REGION Network 211: Transfer P&P Left Clamp WORK
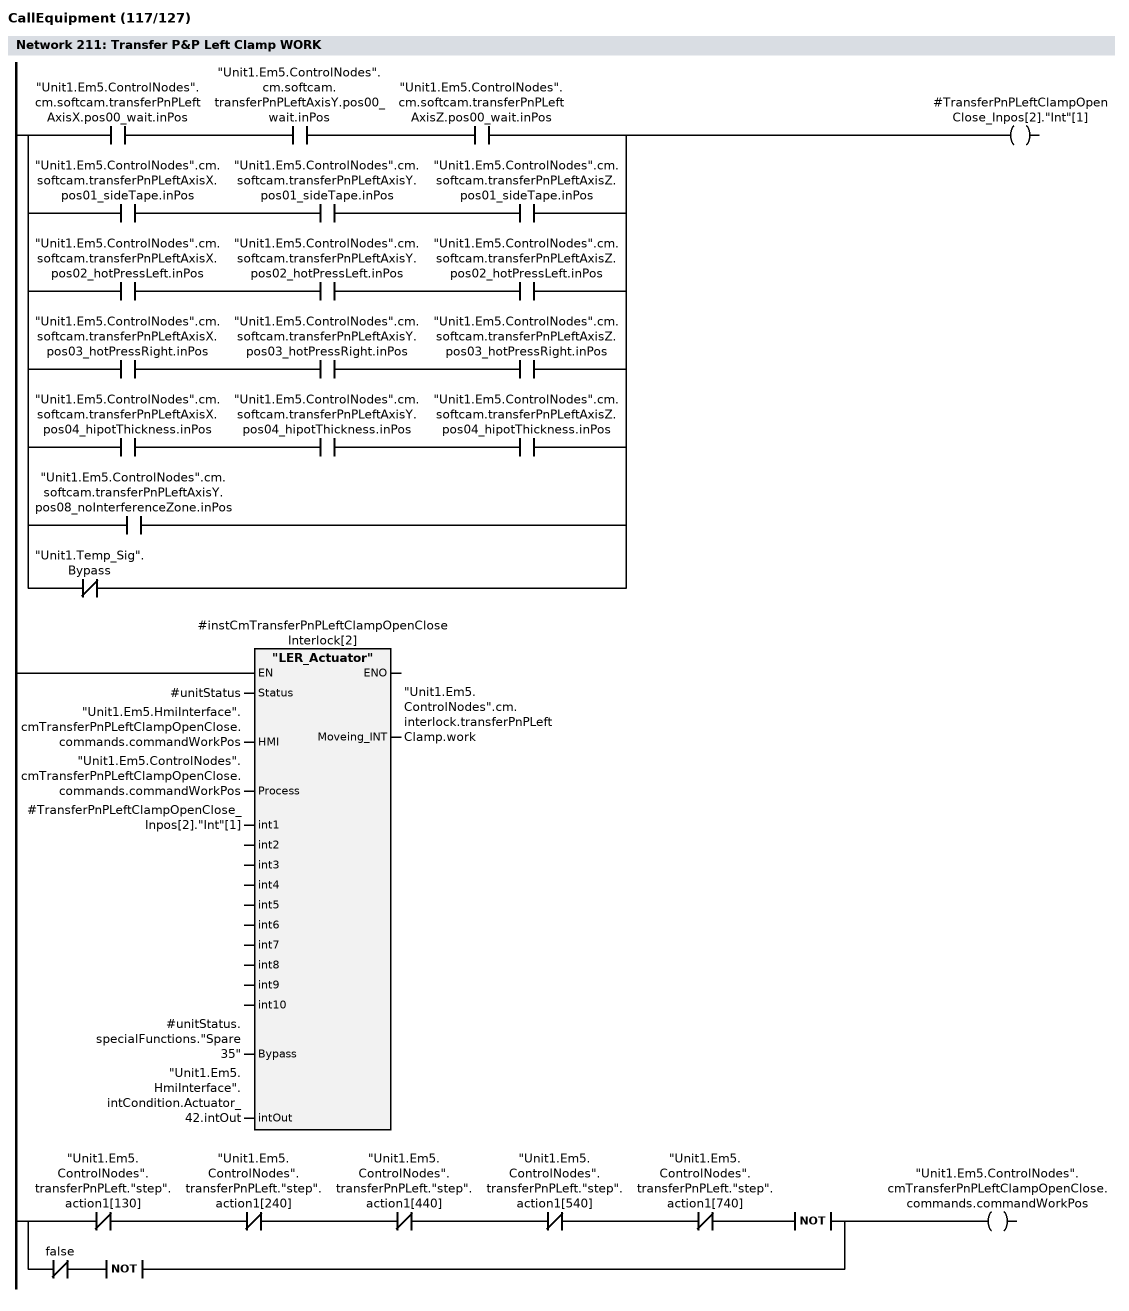
   RUNG wire#powerrail
      Contact( "Unit1.Em5.ControlNodes".cm.softcam.transferPnPLeftAxisX.pos00_wait.inPos )
      Contact( "Unit1.Em5.ControlNodes".cm.softcam.transferPnPLeftAxisY.pos00_wait.inPos )
      Contact( "Unit1.Em5.ControlNodes".cm.softcam.transferPnPLeftAxisZ.pos00_wait.inPos )
      wire#w1
      Coil( #TransferPnPLeftClampOpenClose_Inpos[2]."Int"[1] )
   END_RUNG
   RUNG wire#powerrail
      Contact( "Unit1.Em5.ControlNodes".cm.softcam.transferPnPLeftAxisX.pos01_sideTape.inPos )
      Contact( "Unit1.Em5.ControlNodes".cm.softcam.transferPnPLeftAxisY.pos01_sideTape.inPos )
      Contact( "Unit1.Em5.ControlNodes".cm.softcam.transferPnPLeftAxisZ.pos01_sideTape.inPos )
   END_RUNG wire#w1
   RUNG wire#powerrail
      Contact( "Unit1.Em5.ControlNodes".cm.softcam.transferPnPLeftAxisX.pos02_hotPressLeft.inPos )
      Contact( "Unit1.Em5.ControlNodes".cm.softcam.transferPnPLeftAxisY.pos02_hotPressLeft.inPos )
      Contact( "Unit1.Em5.ControlNodes".cm.softcam.transferPnPLeftAxisZ.pos02_hotPressLeft.inPos )
   END_RUNG wire#w1
   RUNG wire#powerrail
      Contact( "Unit1.Em5.ControlNodes".cm.softcam.transferPnPLeftAxisX.pos03_hotPressRight.inPos )
      Contact( "Unit1.Em5.ControlNodes".cm.softcam.transferPnPLeftAxisY.pos03_hotPressRight.inPos )
      Contact( "Unit1.Em5.ControlNodes".cm.softcam.transferPnPLeftAxisZ.pos03_hotPressRight.inPos )
   END_RUNG wire#w1
   RUNG wire#powerrail
      Contact( "Unit1.Em5.ControlNodes".cm.softcam.transferPnPLeftAxisX.pos04_hipotThickness.inPos )
      Contact( "Unit1.Em5.ControlNodes".cm.softcam.transferPnPLeftAxisY.pos04_hipotThickness.inPos )
      Contact( "Unit1.Em5.ControlNodes".cm.softcam.transferPnPLeftAxisZ.pos04_hipotThickness.inPos )
   END_RUNG wire#w1
   RUNG wire#powerrail
      Contact( "Unit1.Em5.ControlNodes".cm.softcam.transferPnPLeftAxisY.pos08_noInterferenceZone.inPos )
   END_RUNG wire#w1
   RUNG wire#powerrail
      I_Contact( "Unit1.Temp_Sig".Bypass )
   END_RUNG wire#w1
   RUNG wire#powerrail
      #instCmTransferPnPLeftClampOpenCloseInterlock[2](Status := #unitStatus, HMI := "Unit1.Em5.HmiInterface".cmTransferPnPLeftClampOpenClose.commands.commandWorkPos, Process := "Unit1.Em5.ControlNodes".cmTransferPnPLeftClampOpenClose.commands.commandWorkPos, int1 := #TransferPnPLeftClampOpenClose_Inpos[2]."Int"[1], int2 :=, int3 :=, int4 :=, int5 :=, int6 :=, int7 :=, int8 :=, int9 :=, int10 :=, Bypass := #unitStatus.specialFunctions."Spare 35", intOut := "Unit1.Em5.HmiInterface".intCondition.Actuator_42.intOut, Moveing_INT => "Unit1.Em5.ControlNodes".cm.interlock.transferPnPLeftClamp.work)
   END_RUNG
   RUNG wire#powerrail
      I_Contact( "Unit1.Em5.ControlNodes".transferPnPLeft."step".action1[130] )
      I_Contact( "Unit1.Em5.ControlNodes".transferPnPLeft."step".action1[240] )
      I_Contact( "Unit1.Em5.ControlNodes".transferPnPLeft."step".action1[440] )
      I_Contact( "Unit1.Em5.ControlNodes".transferPnPLeft."step".action1[540] )
      I_Contact( "Unit1.Em5.ControlNodes".transferPnPLeft."step".action1[740] )
      Not()
      wire#w2
      Coil( "Unit1.Em5.ControlNodes".cmTransferPnPLeftClampOpenClose.commands.commandWorkPos )
   END_RUNG
   RUNG wire#powerrail
      I_Contact( false )
      Not()
   END_RUNG wire#w2
   // the same network as SCL:
   #TransferPnPLeftClampOpenClose_Inpos[2]."Int"[1] := ("Unit1.Em5.ControlNodes".cm.softcam.transferPnPLeftAxisX.pos00_wait.inPos AND "Unit1.Em5.ControlNodes".cm.softcam.transferPnPLeftAxisY.pos00_wait.inPos AND "Unit1.Em5.ControlNodes".cm.softcam.transferPnPLeftAxisZ.pos00_wait.inPos) OR ("Unit1.Em5.ControlNodes".cm.softcam.transferPnPLeftAxisX.pos01_sideTape.inPos AND "Unit1.Em5.ControlNodes".cm.softcam.transferPnPLeftAxisY.pos01_sideTape.inPos AND "Unit1.Em5.ControlNodes".cm.softcam.transferPnPLeftAxisZ.pos01_sideTape.inPos) OR ("Unit1.Em5.ControlNodes".cm.softcam.transferPnPLeftAxisX.pos02_hotPressLeft.inPos AND "Unit1.Em5.ControlNodes".cm.softcam.transferPnPLeftAxisY.pos02_hotPressLeft.inPos AND "Unit1.Em5.ControlNodes".cm.softcam.transferPnPLeftAxisZ.pos02_hotPressLeft.inPos) OR ("Unit1.Em5.ControlNodes".cm.softcam.transferPnPLeftAxisX.pos03_hotPressRight.inPos AND "Unit1.Em5.ControlNodes".cm.softcam.transferPnPLeftAxisY.pos03_hotPressRight.inPos AND "Unit1.Em5.ControlNodes".cm.softcam.transferPnPLeftAxisZ.pos03_hotPressRight.inPos) OR ("Unit1.Em5.ControlNodes".cm.softcam.transferPnPLeftAxisX.pos04_hipotThickness.inPos AND "Unit1.Em5.ControlNodes".cm.softcam.transferPnPLeftAxisY.pos04_hipotThickness.inPos AND "Unit1.Em5.ControlNodes".cm.softcam.transferPnPLeftAxisZ.pos04_hipotThickness.inPos) OR "Unit1.Em5.ControlNodes".cm.softcam.transferPnPLeftAxisY.pos08_noInterferenceZone.inPos OR NOT "Unit1.Temp_Sig".Bypass;
   #instCmTransferPnPLeftClampOpenCloseInterlock[2](Status := #unitStatus,   // "LER_Actuator"
                           HMI := "Unit1.Em5.HmiInterface".cmTransferPnPLeftClampOpenClose.commands.commandWorkPos,
                           Process := "Unit1.Em5.ControlNodes".cmTransferPnPLeftClampOpenClose.commands.commandWorkPos,
                           int1 := #TransferPnPLeftClampOpenClose_Inpos[2]."Int"[1],
                           Bypass := #unitStatus.specialFunctions."Spare 35",
                           intOut := "Unit1.Em5.HmiInterface".intCondition.Actuator_42.intOut,
                           Moveing_INT => "Unit1.Em5.ControlNodes".cm.interlock.transferPnPLeftClamp.work);
   "Unit1.Em5.ControlNodes".cmTransferPnPLeftClampOpenClose.commands.commandWorkPos := NOT (NOT "Unit1.Em5.ControlNodes".transferPnPLeft."step".action1[130] AND NOT "Unit1.Em5.ControlNodes".transferPnPLeft."step".action1[240] AND NOT "Unit1.Em5.ControlNodes".transferPnPLeft."step".action1[440] AND NOT "Unit1.Em5.ControlNodes".transferPnPLeft."step".action1[540] AND NOT "Unit1.Em5.ControlNodes".transferPnPLeft."step".action1[740]) OR NOT (NOT false);
END_REGION

REGION Network 212: Call CM Transfer P&P Left Clamp Open/Close (LBC_TwoWayActuator)
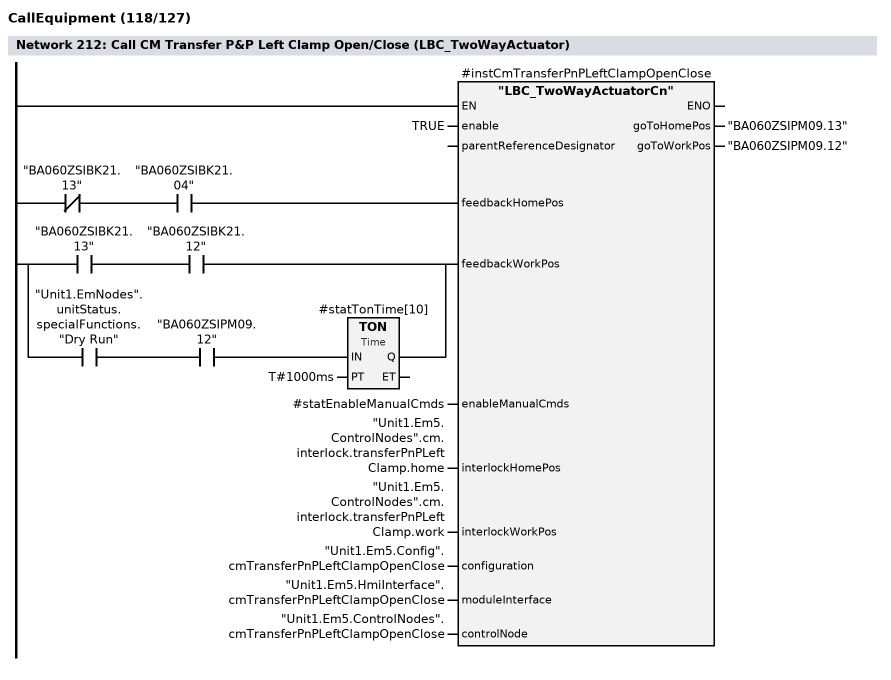
   RUNG wire#powerrail
      #instCmTransferPnPLeftClampOpenClose(feedbackHomePos := wire#w1, feedbackWorkPos := wire#w2, enable := TRUE, parentReferenceDesignator :=, enableManualCmds := #statEnableManualCmds, interlockHomePos := "Unit1.Em5.ControlNodes".cm.interlock.transferPnPLeftClamp.home, interlockWorkPos := "Unit1.Em5.ControlNodes".cm.interlock.transferPnPLeftClamp.work, configuration := "Unit1.Em5.Config".cmTransferPnPLeftClampOpenClose, moduleInterface := "Unit1.Em5.HmiInterface".cmTransferPnPLeftClampOpenClose, controlNode := "Unit1.Em5.ControlNodes".cmTransferPnPLeftClampOpenClose, goToHomePos => "BA060ZSIPM09.13", goToWorkPos => "BA060ZSIPM09.12")
   END_RUNG
   RUNG wire#powerrail
      I_Contact( "BA060ZSIBK21.13" )
      Contact( "BA060ZSIBK21.04" )
   END_RUNG wire#w1
   RUNG wire#powerrail
      Contact( "BA060ZSIBK21.13" )
      Contact( "BA060ZSIBK21.12" )
   END_RUNG wire#w2
   RUNG wire#powerrail
      Contact( "Unit1.EmNodes".unitStatus.specialFunctions."Dry Run" )
      Contact( "BA060ZSIPM09.12" )
      { S7_Templates := "time_type := Time" } #statTonTime[10].TON(pt := T#1000ms, et =>)
   END_RUNG wire#w2
   // the same network as SCL:
   #statTonTime[10].TON(IN := "Unit1.EmNodes".unitStatus.specialFunctions."Dry Run" AND "BA060ZSIPM09.12",
                        PT := T#1000ms);
   #instCmTransferPnPLeftClampOpenClose(enable := TRUE,   // "LBC_TwoWayActuatorCn"
                           feedbackHomePos := NOT "BA060ZSIBK21.13" AND "BA060ZSIBK21.04",
                           feedbackWorkPos := ("BA060ZSIBK21.13" AND "BA060ZSIBK21.12") OR #statTonTime[10].Q,
                           enableManualCmds := #statEnableManualCmds,
                           interlockHomePos := "Unit1.Em5.ControlNodes".cm.interlock.transferPnPLeftClamp.home,
                           interlockWorkPos := "Unit1.Em5.ControlNodes".cm.interlock.transferPnPLeftClamp.work,
                           configuration := "Unit1.Em5.Config".cmTransferPnPLeftClampOpenClose,
                           moduleInterface := "Unit1.Em5.HmiInterface".cmTransferPnPLeftClampOpenClose,
                           controlNode := "Unit1.Em5.ControlNodes".cmTransferPnPLeftClampOpenClose,
                           goToHomePos => "BA060ZSIPM09.13",
                           goToWorkPos => "BA060ZSIPM09.12");
END_REGION

REGION Network 214: Transfer P&P Right Clamp HOME
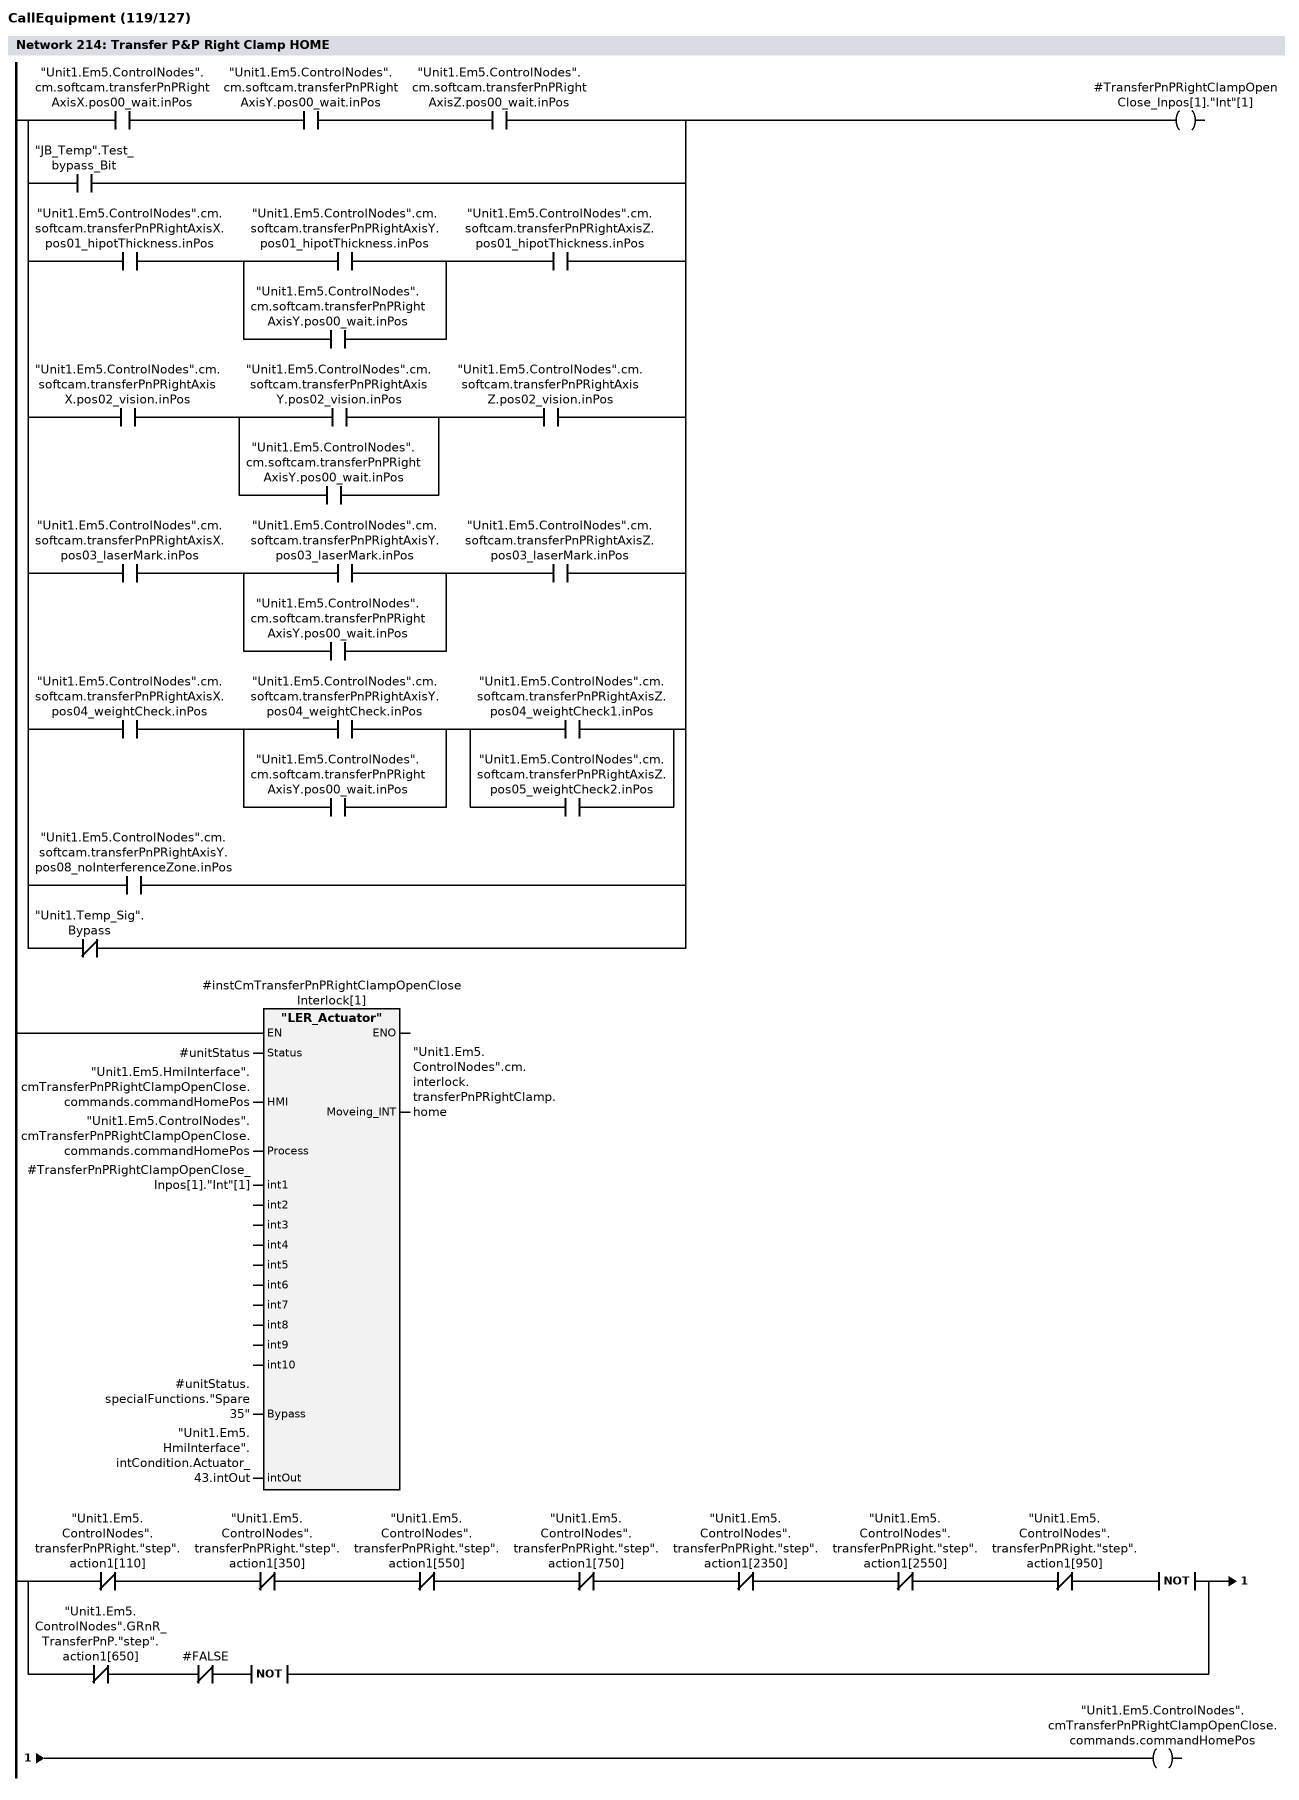
   RUNG wire#powerrail
      Contact( "Unit1.Em5.ControlNodes".cm.softcam.transferPnPRightAxisX.pos00_wait.inPos )
      Contact( "Unit1.Em5.ControlNodes".cm.softcam.transferPnPRightAxisY.pos00_wait.inPos )
      Contact( "Unit1.Em5.ControlNodes".cm.softcam.transferPnPRightAxisZ.pos00_wait.inPos )
      wire#w1
      Coil( #TransferPnPRightClampOpenClose_Inpos[1]."Int"[1] )
   END_RUNG
   RUNG wire#powerrail
      Contact( "JB_Temp".Test_bypass_Bit )
   END_RUNG wire#w1
   RUNG wire#powerrail
      Contact( "Unit1.Em5.ControlNodes".cm.softcam.transferPnPRightAxisX.pos01_hipotThickness.inPos )
      wire#w2
      Contact( "Unit1.Em5.ControlNodes".cm.softcam.transferPnPRightAxisY.pos01_hipotThickness.inPos )
      wire#w3
      Contact( "Unit1.Em5.ControlNodes".cm.softcam.transferPnPRightAxisZ.pos01_hipotThickness.inPos )
   END_RUNG wire#w1
   RUNG wire#w2
      Contact( "Unit1.Em5.ControlNodes".cm.softcam.transferPnPRightAxisY.pos00_wait.inPos )
   END_RUNG wire#w3
   RUNG wire#powerrail
      Contact( "Unit1.Em5.ControlNodes".cm.softcam.transferPnPRightAxisX.pos02_vision.inPos )
      wire#w4
      Contact( "Unit1.Em5.ControlNodes".cm.softcam.transferPnPRightAxisY.pos02_vision.inPos )
      wire#w5
      Contact( "Unit1.Em5.ControlNodes".cm.softcam.transferPnPRightAxisZ.pos02_vision.inPos )
   END_RUNG wire#w1
   RUNG wire#w4
      Contact( "Unit1.Em5.ControlNodes".cm.softcam.transferPnPRightAxisY.pos00_wait.inPos )
   END_RUNG wire#w5
   RUNG wire#powerrail
      Contact( "Unit1.Em5.ControlNodes".cm.softcam.transferPnPRightAxisX.pos03_laserMark.inPos )
      wire#w6
      Contact( "Unit1.Em5.ControlNodes".cm.softcam.transferPnPRightAxisY.pos03_laserMark.inPos )
      wire#w7
      Contact( "Unit1.Em5.ControlNodes".cm.softcam.transferPnPRightAxisZ.pos03_laserMark.inPos )
   END_RUNG wire#w1
   RUNG wire#w6
      Contact( "Unit1.Em5.ControlNodes".cm.softcam.transferPnPRightAxisY.pos00_wait.inPos )
   END_RUNG wire#w7
   RUNG wire#powerrail
      Contact( "Unit1.Em5.ControlNodes".cm.softcam.transferPnPRightAxisX.pos04_weightCheck.inPos )
      wire#w8
      Contact( "Unit1.Em5.ControlNodes".cm.softcam.transferPnPRightAxisY.pos04_weightCheck.inPos )
      wire#w9
      Contact( "Unit1.Em5.ControlNodes".cm.softcam.transferPnPRightAxisZ.pos04_weightCheck1.inPos )
   END_RUNG wire#w1
   RUNG wire#w8
      Contact( "Unit1.Em5.ControlNodes".cm.softcam.transferPnPRightAxisY.pos00_wait.inPos )
   END_RUNG wire#w9
   RUNG wire#w9
      Contact( "Unit1.Em5.ControlNodes".cm.softcam.transferPnPRightAxisZ.pos05_weightCheck2.inPos )
   END_RUNG wire#w1
   RUNG wire#powerrail
      Contact( "Unit1.Em5.ControlNodes".cm.softcam.transferPnPRightAxisY.pos08_noInterferenceZone.inPos )
   END_RUNG wire#w1
   RUNG wire#powerrail
      I_Contact( "Unit1.Temp_Sig".Bypass )
   END_RUNG wire#w1
   RUNG wire#powerrail
      #instCmTransferPnPRightClampOpenCloseInterlock[1](Status := #unitStatus, HMI := "Unit1.Em5.HmiInterface".cmTransferPnPRightClampOpenClose.commands.commandHomePos, Process := "Unit1.Em5.ControlNodes".cmTransferPnPRightClampOpenClose.commands.commandHomePos, int1 := #TransferPnPRightClampOpenClose_Inpos[1]."Int"[1], int2 :=, int3 :=, int4 :=, int5 :=, int6 :=, int7 :=, int8 :=, int9 :=, int10 :=, Bypass := #unitStatus.specialFunctions."Spare 35", intOut := "Unit1.Em5.HmiInterface".intCondition.Actuator_43.intOut, Moveing_INT => "Unit1.Em5.ControlNodes".cm.interlock.transferPnPRightClamp.home)
   END_RUNG
   RUNG wire#powerrail
      I_Contact( "Unit1.Em5.ControlNodes".transferPnPRight."step".action1[110] )
      I_Contact( "Unit1.Em5.ControlNodes".transferPnPRight."step".action1[350] )
      I_Contact( "Unit1.Em5.ControlNodes".transferPnPRight."step".action1[550] )
      I_Contact( "Unit1.Em5.ControlNodes".transferPnPRight."step".action1[750] )
      I_Contact( "Unit1.Em5.ControlNodes".transferPnPRight."step".action1[2350] )
      I_Contact( "Unit1.Em5.ControlNodes".transferPnPRight."step".action1[2550] )
      I_Contact( "Unit1.Em5.ControlNodes".transferPnPRight."step".action1[950] )
      Not()
      wire#w10
      Coil( "Unit1.Em5.ControlNodes".cmTransferPnPRightClampOpenClose.commands.commandHomePos )
   END_RUNG
   RUNG wire#powerrail
      I_Contact( "Unit1.Em5.ControlNodes".GRnR_TransferPnP."step".action1[650] )
      I_Contact( #FALSE )
      Not()
   END_RUNG wire#w10
   // the same network as SCL:
   #TransferPnPRightClampOpenClose_Inpos[1]."Int"[1] := ("Unit1.Em5.ControlNodes".cm.softcam.transferPnPRightAxisX.pos00_wait.inPos AND "Unit1.Em5.ControlNodes".cm.softcam.transferPnPRightAxisY.pos00_wait.inPos AND "Unit1.Em5.ControlNodes".cm.softcam.transferPnPRightAxisZ.pos00_wait.inPos) OR "JB_Temp".Test_bypass_Bit OR ("Unit1.Em5.ControlNodes".cm.softcam.transferPnPRightAxisX.pos01_hipotThickness.inPos AND ("Unit1.Em5.ControlNodes".cm.softcam.transferPnPRightAxisY.pos01_hipotThickness.inPos OR "Unit1.Em5.ControlNodes".cm.softcam.transferPnPRightAxisY.pos00_wait.inPos) AND "Unit1.Em5.ControlNodes".cm.softcam.transferPnPRightAxisZ.pos01_hipotThickness.inPos) OR ("Unit1.Em5.ControlNodes".cm.softcam.transferPnPRightAxisX.pos02_vision.inPos AND ("Unit1.Em5.ControlNodes".cm.softcam.transferPnPRightAxisY.pos02_vision.inPos OR "Unit1.Em5.ControlNodes".cm.softcam.transferPnPRightAxisY.pos00_wait.inPos) AND "Unit1.Em5.ControlNodes".cm.softcam.transferPnPRightAxisZ.pos02_vision.inPos) OR ("Unit1.Em5.ControlNodes".cm.softcam.transferPnPRightAxisX.pos03_laserMark.inPos AND ("Unit1.Em5.ControlNodes".cm.softcam.transferPnPRightAxisY.pos03_laserMark.inPos OR "Unit1.Em5.ControlNodes".cm.softcam.transferPnPRightAxisY.pos00_wait.inPos) AND "Unit1.Em5.ControlNodes".cm.softcam.transferPnPRightAxisZ.pos03_laserMark.inPos) OR ("Unit1.Em5.ControlNodes".cm.softcam.transferPnPRightAxisX.pos04_weightCheck.inPos AND ("Unit1.Em5.ControlNodes".cm.softcam.transferPnPRightAxisY.pos04_weightCheck.inPos OR "Unit1.Em5.ControlNodes".cm.softcam.transferPnPRightAxisY.pos00_wait.inPos) AND ("Unit1.Em5.ControlNodes".cm.softcam.transferPnPRightAxisZ.pos04_weightCheck1.inPos OR "Unit1.Em5.ControlNodes".cm.softcam.transferPnPRightAxisZ.pos05_weightCheck2.inPos)) OR "Unit1.Em5.ControlNodes".cm.softcam.transferPnPRightAxisY.pos08_noInterferenceZone.inPos OR NOT "Unit1.Temp_Sig".Bypass;
   #instCmTransferPnPRightClampOpenCloseInterlock[1](Status := #unitStatus,   // "LER_Actuator"
                           HMI := "Unit1.Em5.HmiInterface".cmTransferPnPRightClampOpenClose.commands.commandHomePos,
                           Process := "Unit1.Em5.ControlNodes".cmTransferPnPRightClampOpenClose.commands.commandHomePos,
                           int1 := #TransferPnPRightClampOpenClose_Inpos[1]."Int"[1],
                           Bypass := #unitStatus.specialFunctions."Spare 35",
                           intOut := "Unit1.Em5.HmiInterface".intCondition.Actuator_43.intOut,
                           Moveing_INT => "Unit1.Em5.ControlNodes".cm.interlock.transferPnPRightClamp.home);
   "Unit1.Em5.ControlNodes".cmTransferPnPRightClampOpenClose.commands.commandHomePos := NOT (NOT "Unit1.Em5.ControlNodes".transferPnPRight."step".action1[110] AND NOT "Unit1.Em5.ControlNodes".transferPnPRight."step".action1[350] AND NOT "Unit1.Em5.ControlNodes".transferPnPRight."step".action1[550] AND NOT "Unit1.Em5.ControlNodes".transferPnPRight."step".action1[750] AND NOT "Unit1.Em5.ControlNodes".transferPnPRight."step".action1[2350] AND NOT "Unit1.Em5.ControlNodes".transferPnPRight."step".action1[2550] AND NOT "Unit1.Em5.ControlNodes".transferPnPRight."step".action1[950]) OR NOT (NOT "Unit1.Em5.ControlNodes".GRnR_TransferPnP."step".action1[650] AND NOT #FALSE);
END_REGION

REGION Network 215: Transfer P&P Right Clamp WORK
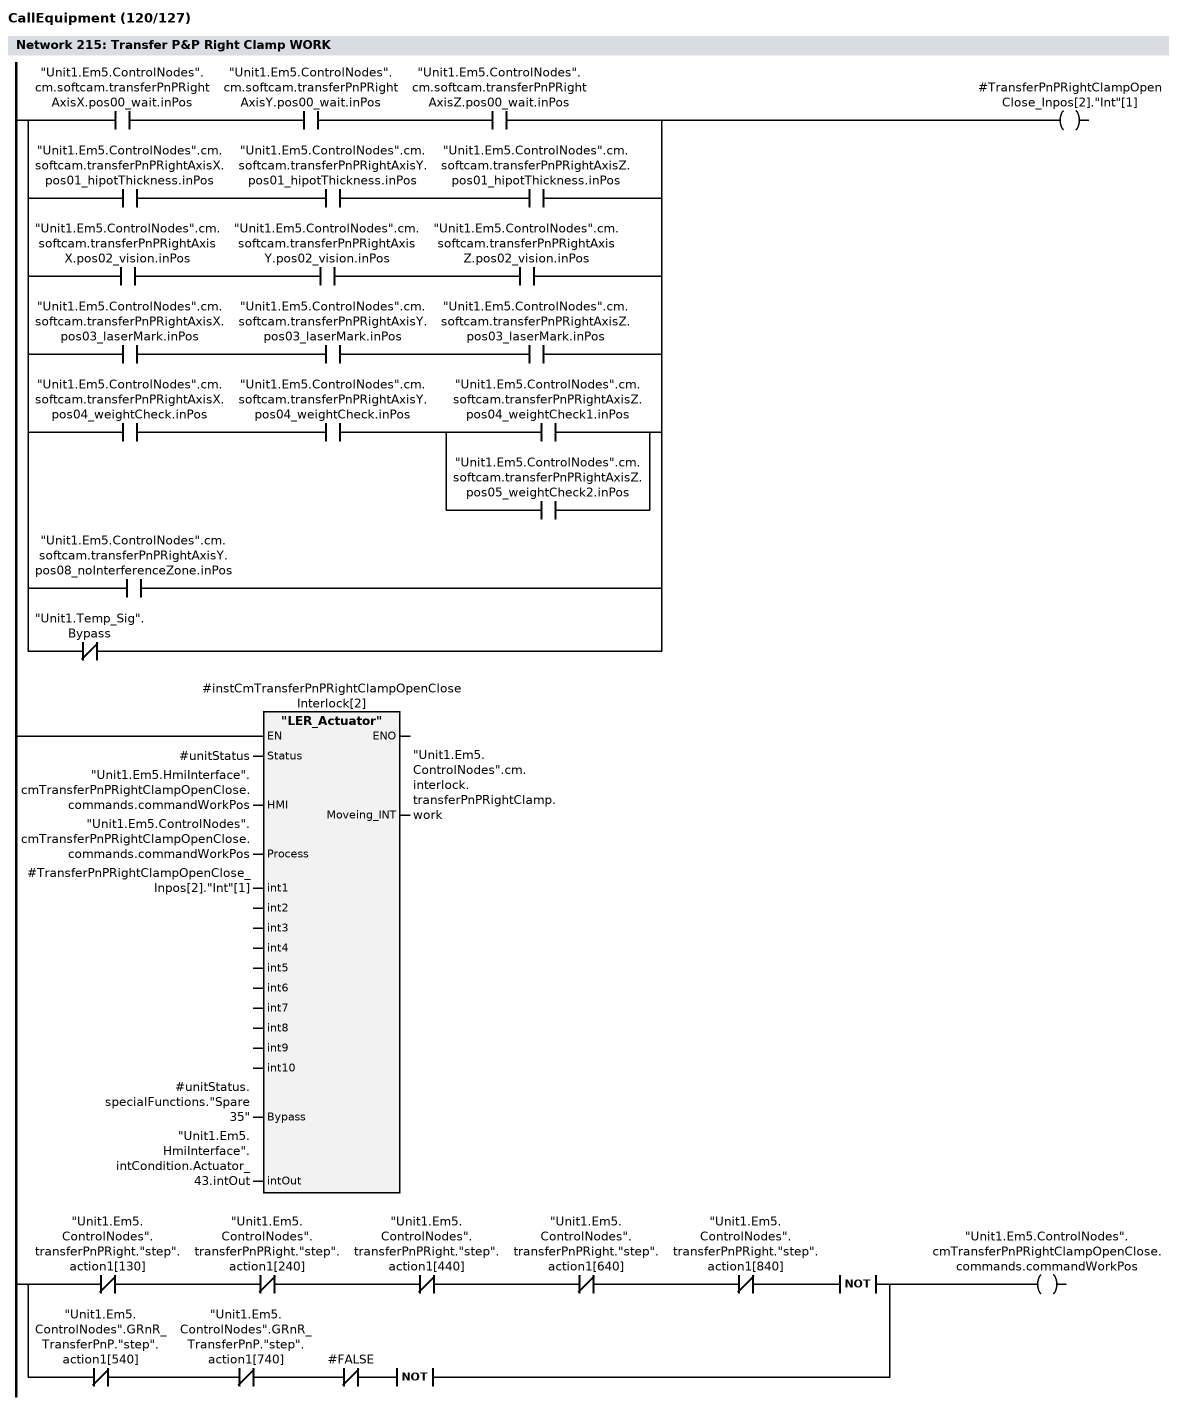
   RUNG wire#powerrail
      Contact( "Unit1.Em5.ControlNodes".cm.softcam.transferPnPRightAxisX.pos00_wait.inPos )
      Contact( "Unit1.Em5.ControlNodes".cm.softcam.transferPnPRightAxisY.pos00_wait.inPos )
      Contact( "Unit1.Em5.ControlNodes".cm.softcam.transferPnPRightAxisZ.pos00_wait.inPos )
      wire#w1
      Coil( #TransferPnPRightClampOpenClose_Inpos[2]."Int"[1] )
   END_RUNG
   RUNG wire#powerrail
      Contact( "Unit1.Em5.ControlNodes".cm.softcam.transferPnPRightAxisX.pos01_hipotThickness.inPos )
      Contact( "Unit1.Em5.ControlNodes".cm.softcam.transferPnPRightAxisY.pos01_hipotThickness.inPos )
      Contact( "Unit1.Em5.ControlNodes".cm.softcam.transferPnPRightAxisZ.pos01_hipotThickness.inPos )
   END_RUNG wire#w1
   RUNG wire#powerrail
      Contact( "Unit1.Em5.ControlNodes".cm.softcam.transferPnPRightAxisX.pos02_vision.inPos )
      Contact( "Unit1.Em5.ControlNodes".cm.softcam.transferPnPRightAxisY.pos02_vision.inPos )
      Contact( "Unit1.Em5.ControlNodes".cm.softcam.transferPnPRightAxisZ.pos02_vision.inPos )
   END_RUNG wire#w1
   RUNG wire#powerrail
      Contact( "Unit1.Em5.ControlNodes".cm.softcam.transferPnPRightAxisX.pos03_laserMark.inPos )
      Contact( "Unit1.Em5.ControlNodes".cm.softcam.transferPnPRightAxisY.pos03_laserMark.inPos )
      Contact( "Unit1.Em5.ControlNodes".cm.softcam.transferPnPRightAxisZ.pos03_laserMark.inPos )
   END_RUNG wire#w1
   RUNG wire#powerrail
      Contact( "Unit1.Em5.ControlNodes".cm.softcam.transferPnPRightAxisX.pos04_weightCheck.inPos )
      Contact( "Unit1.Em5.ControlNodes".cm.softcam.transferPnPRightAxisY.pos04_weightCheck.inPos )
      wire#w2
      Contact( "Unit1.Em5.ControlNodes".cm.softcam.transferPnPRightAxisZ.pos04_weightCheck1.inPos )
   END_RUNG wire#w1
   RUNG wire#w2
      Contact( "Unit1.Em5.ControlNodes".cm.softcam.transferPnPRightAxisZ.pos05_weightCheck2.inPos )
   END_RUNG wire#w1
   RUNG wire#powerrail
      Contact( "Unit1.Em5.ControlNodes".cm.softcam.transferPnPRightAxisY.pos08_noInterferenceZone.inPos )
   END_RUNG wire#w1
   RUNG wire#powerrail
      I_Contact( "Unit1.Temp_Sig".Bypass )
   END_RUNG wire#w1
   RUNG wire#powerrail
      #instCmTransferPnPRightClampOpenCloseInterlock[2](Status := #unitStatus, HMI := "Unit1.Em5.HmiInterface".cmTransferPnPRightClampOpenClose.commands.commandWorkPos, Process := "Unit1.Em5.ControlNodes".cmTransferPnPRightClampOpenClose.commands.commandWorkPos, int1 := #TransferPnPRightClampOpenClose_Inpos[2]."Int"[1], int2 :=, int3 :=, int4 :=, int5 :=, int6 :=, int7 :=, int8 :=, int9 :=, int10 :=, Bypass := #unitStatus.specialFunctions."Spare 35", intOut := "Unit1.Em5.HmiInterface".intCondition.Actuator_43.intOut, Moveing_INT => "Unit1.Em5.ControlNodes".cm.interlock.transferPnPRightClamp.work)
   END_RUNG
   RUNG wire#powerrail
      I_Contact( "Unit1.Em5.ControlNodes".transferPnPRight."step".action1[130] )
      I_Contact( "Unit1.Em5.ControlNodes".transferPnPRight."step".action1[240] )
      I_Contact( "Unit1.Em5.ControlNodes".transferPnPRight."step".action1[440] )
      I_Contact( "Unit1.Em5.ControlNodes".transferPnPRight."step".action1[640] )
      I_Contact( "Unit1.Em5.ControlNodes".transferPnPRight."step".action1[840] )
      Not()
      wire#w3
      Coil( "Unit1.Em5.ControlNodes".cmTransferPnPRightClampOpenClose.commands.commandWorkPos )
   END_RUNG
   RUNG wire#powerrail
      I_Contact( "Unit1.Em5.ControlNodes".GRnR_TransferPnP."step".action1[540] )
      I_Contact( "Unit1.Em5.ControlNodes".GRnR_TransferPnP."step".action1[740] )
      I_Contact( #FALSE )
      Not()
   END_RUNG wire#w3
   // the same network as SCL:
   #TransferPnPRightClampOpenClose_Inpos[2]."Int"[1] := ("Unit1.Em5.ControlNodes".cm.softcam.transferPnPRightAxisX.pos00_wait.inPos AND "Unit1.Em5.ControlNodes".cm.softcam.transferPnPRightAxisY.pos00_wait.inPos AND "Unit1.Em5.ControlNodes".cm.softcam.transferPnPRightAxisZ.pos00_wait.inPos) OR ("Unit1.Em5.ControlNodes".cm.softcam.transferPnPRightAxisX.pos01_hipotThickness.inPos AND "Unit1.Em5.ControlNodes".cm.softcam.transferPnPRightAxisY.pos01_hipotThickness.inPos AND "Unit1.Em5.ControlNodes".cm.softcam.transferPnPRightAxisZ.pos01_hipotThickness.inPos) OR ("Unit1.Em5.ControlNodes".cm.softcam.transferPnPRightAxisX.pos02_vision.inPos AND "Unit1.Em5.ControlNodes".cm.softcam.transferPnPRightAxisY.pos02_vision.inPos AND "Unit1.Em5.ControlNodes".cm.softcam.transferPnPRightAxisZ.pos02_vision.inPos) OR ("Unit1.Em5.ControlNodes".cm.softcam.transferPnPRightAxisX.pos03_laserMark.inPos AND "Unit1.Em5.ControlNodes".cm.softcam.transferPnPRightAxisY.pos03_laserMark.inPos AND "Unit1.Em5.ControlNodes".cm.softcam.transferPnPRightAxisZ.pos03_laserMark.inPos) OR ("Unit1.Em5.ControlNodes".cm.softcam.transferPnPRightAxisX.pos04_weightCheck.inPos AND "Unit1.Em5.ControlNodes".cm.softcam.transferPnPRightAxisY.pos04_weightCheck.inPos AND ("Unit1.Em5.ControlNodes".cm.softcam.transferPnPRightAxisZ.pos04_weightCheck1.inPos OR "Unit1.Em5.ControlNodes".cm.softcam.transferPnPRightAxisZ.pos05_weightCheck2.inPos)) OR "Unit1.Em5.ControlNodes".cm.softcam.transferPnPRightAxisY.pos08_noInterferenceZone.inPos OR NOT "Unit1.Temp_Sig".Bypass;
   #instCmTransferPnPRightClampOpenCloseInterlock[2](Status := #unitStatus,   // "LER_Actuator"
                           HMI := "Unit1.Em5.HmiInterface".cmTransferPnPRightClampOpenClose.commands.commandWorkPos,
                           Process := "Unit1.Em5.ControlNodes".cmTransferPnPRightClampOpenClose.commands.commandWorkPos,
                           int1 := #TransferPnPRightClampOpenClose_Inpos[2]."Int"[1],
                           Bypass := #unitStatus.specialFunctions."Spare 35",
                           intOut := "Unit1.Em5.HmiInterface".intCondition.Actuator_43.intOut,
                           Moveing_INT => "Unit1.Em5.ControlNodes".cm.interlock.transferPnPRightClamp.work);
   "Unit1.Em5.ControlNodes".cmTransferPnPRightClampOpenClose.commands.commandWorkPos := NOT (NOT "Unit1.Em5.ControlNodes".transferPnPRight."step".action1[130] AND NOT "Unit1.Em5.ControlNodes".transferPnPRight."step".action1[240] AND NOT "Unit1.Em5.ControlNodes".transferPnPRight."step".action1[440] AND NOT "Unit1.Em5.ControlNodes".transferPnPRight."step".action1[640] AND NOT "Unit1.Em5.ControlNodes".transferPnPRight."step".action1[840]) OR NOT (NOT "Unit1.Em5.ControlNodes".GRnR_TransferPnP."step".action1[540] AND NOT "Unit1.Em5.ControlNodes".GRnR_TransferPnP."step".action1[740] AND NOT #FALSE);
END_REGION

REGION Network 216: Call CM Transfer P&P Right Clamp Open/Close (LBC_TwoWayActuator)
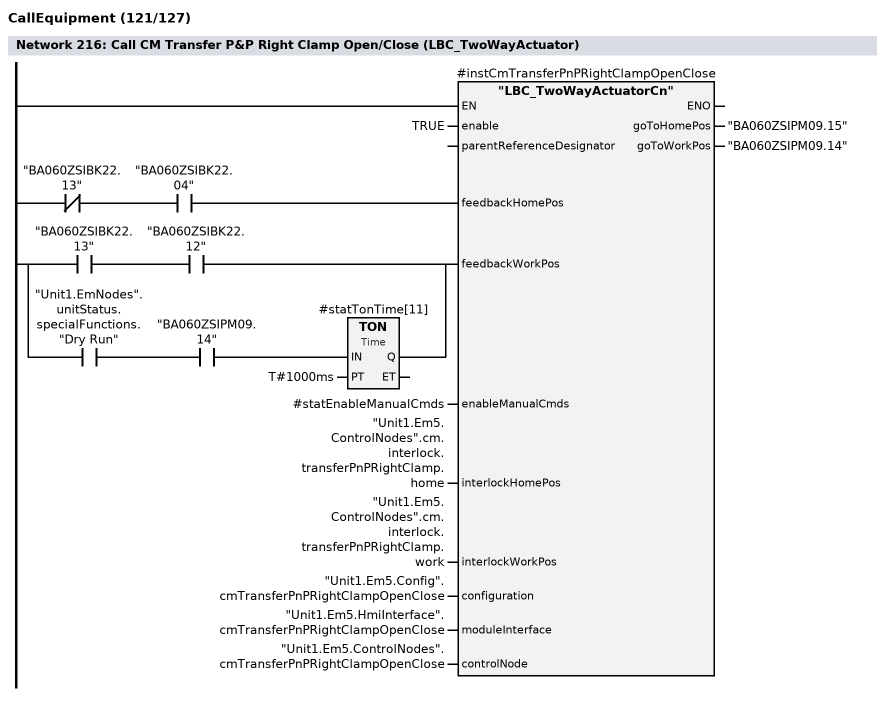
   RUNG wire#powerrail
      #instCmTransferPnPRightClampOpenClose(feedbackHomePos := wire#w1, feedbackWorkPos := wire#w2, enable := TRUE, parentReferenceDesignator :=, enableManualCmds := #statEnableManualCmds, interlockHomePos := "Unit1.Em5.ControlNodes".cm.interlock.transferPnPRightClamp.home, interlockWorkPos := "Unit1.Em5.ControlNodes".cm.interlock.transferPnPRightClamp.work, configuration := "Unit1.Em5.Config".cmTransferPnPRightClampOpenClose, moduleInterface := "Unit1.Em5.HmiInterface".cmTransferPnPRightClampOpenClose, controlNode := "Unit1.Em5.ControlNodes".cmTransferPnPRightClampOpenClose, goToHomePos => "BA060ZSIPM09.15", goToWorkPos => "BA060ZSIPM09.14")
   END_RUNG
   RUNG wire#powerrail
      I_Contact( "BA060ZSIBK22.13" )
      Contact( "BA060ZSIBK22.04" )
   END_RUNG wire#w1
   RUNG wire#powerrail
      Contact( "BA060ZSIBK22.13" )
      Contact( "BA060ZSIBK22.12" )
   END_RUNG wire#w2
   RUNG wire#powerrail
      Contact( "Unit1.EmNodes".unitStatus.specialFunctions."Dry Run" )
      Contact( "BA060ZSIPM09.14" )
      { S7_Templates := "time_type := Time" } #statTonTime[11].TON(pt := T#1000ms, et =>)
   END_RUNG wire#w2
   // the same network as SCL:
   #statTonTime[11].TON(IN := "Unit1.EmNodes".unitStatus.specialFunctions."Dry Run" AND "BA060ZSIPM09.14",
                        PT := T#1000ms);
   #instCmTransferPnPRightClampOpenClose(enable := TRUE,   // "LBC_TwoWayActuatorCn"
                           feedbackHomePos := NOT "BA060ZSIBK22.13" AND "BA060ZSIBK22.04",
                           feedbackWorkPos := ("BA060ZSIBK22.13" AND "BA060ZSIBK22.12") OR #statTonTime[11].Q,
                           enableManualCmds := #statEnableManualCmds,
                           interlockHomePos := "Unit1.Em5.ControlNodes".cm.interlock.transferPnPRightClamp.home,
                           interlockWorkPos := "Unit1.Em5.ControlNodes".cm.interlock.transferPnPRightClamp.work,
                           configuration := "Unit1.Em5.Config".cmTransferPnPRightClampOpenClose,
                           moduleInterface := "Unit1.Em5.HmiInterface".cmTransferPnPRightClampOpenClose,
                           controlNode := "Unit1.Em5.ControlNodes".cmTransferPnPRightClampOpenClose,
                           goToHomePos => "BA060ZSIPM09.15",
                           goToWorkPos => "BA060ZSIPM09.14");
END_REGION

REGION Network 218: ******************** Feedback to Unit ********************
END_REGION

REGION Network 219: Determine StateComplete (SC) in Mode Production
   // Conditions for the Equipment Modules "stateComplete" feedback to the unit. This feedback is given when the task in for the respective state is complete.
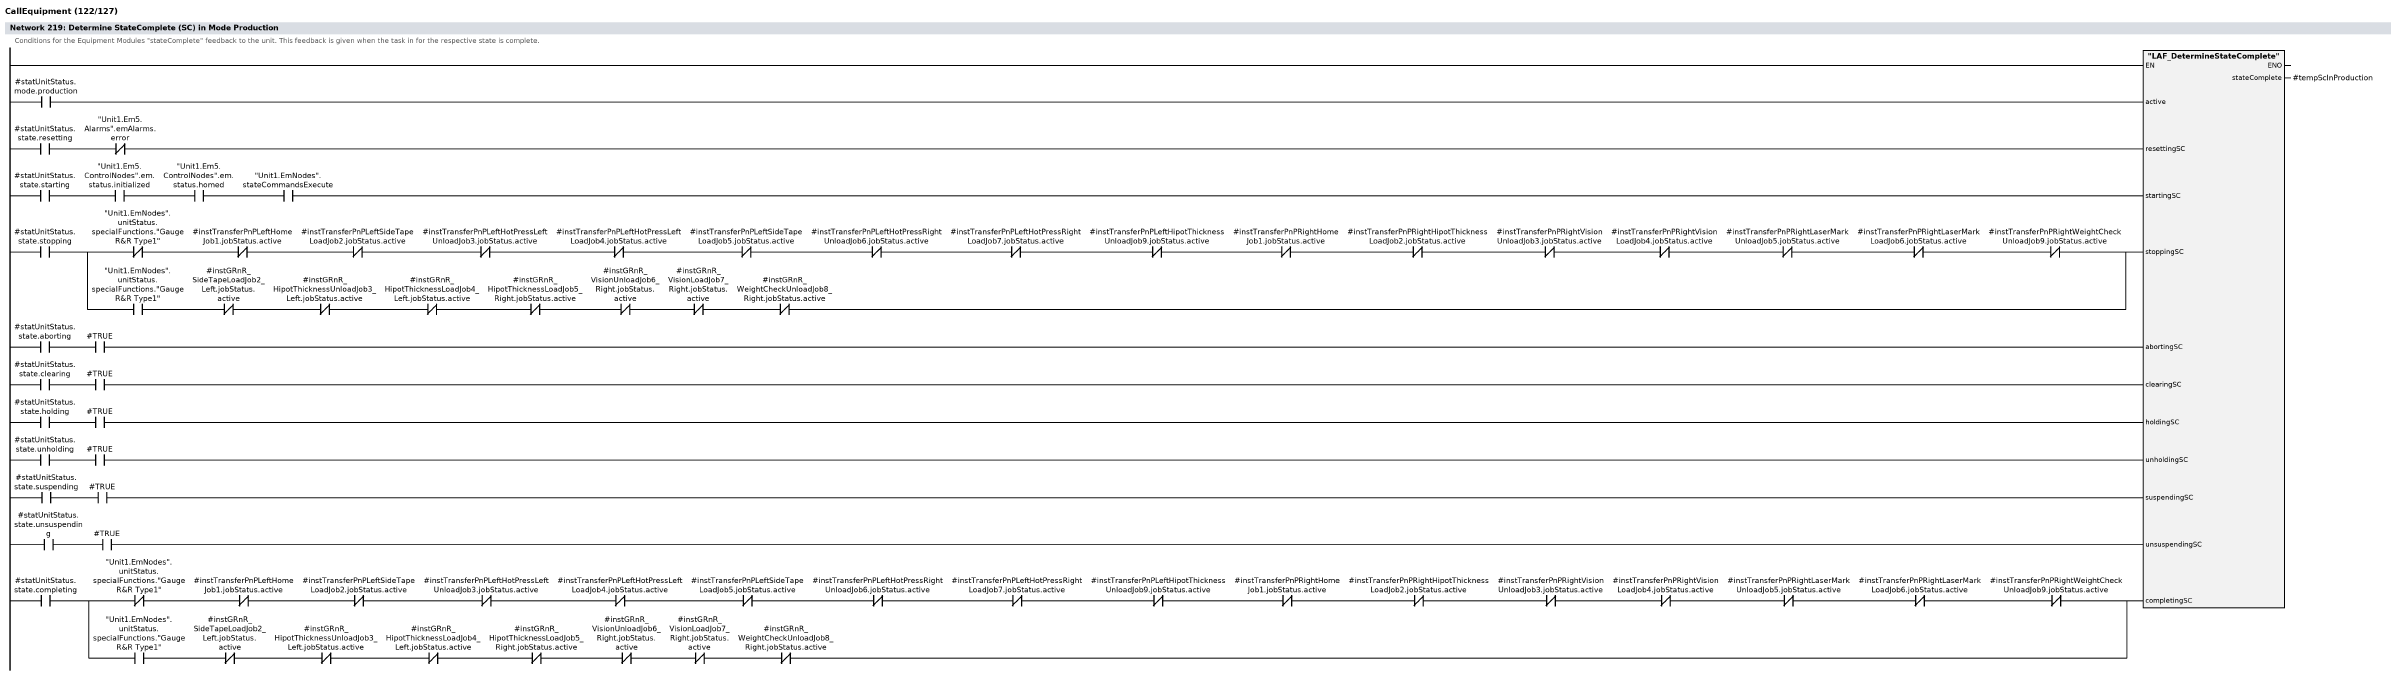
   RUNG wire#powerrail
      "LAF_DetermineStateComplete"(active := wire#w1, resettingSC := wire#w2, startingSC := wire#w3, stoppingSC := wire#w5, abortingSC := wire#w6, clearingSC := wire#w7, holdingSC := wire#w8, unholdingSC := wire#w9, suspendingSC := wire#w10, unsuspendingSC := wire#w11, completingSC := wire#w13, stateComplete => #tempScInProduction)
   END_RUNG
   RUNG wire#powerrail
      Contact( #statUnitStatus.mode.production )
   END_RUNG wire#w1
   RUNG wire#powerrail
      Contact( #statUnitStatus.state.resetting )
      I_Contact( "Unit1.Em5.Alarms".emAlarms.error )
   END_RUNG wire#w2
   RUNG wire#powerrail
      Contact( #statUnitStatus.state.starting )
      Contact( "Unit1.Em5.ControlNodes".em.status.initialized )
      Contact( "Unit1.Em5.ControlNodes".em.status.homed )
      Contact( "Unit1.EmNodes".stateCommandsExecute )
   END_RUNG wire#w3
   RUNG wire#powerrail
      Contact( #statUnitStatus.state.stopping )
      wire#w4
      I_Contact( "Unit1.EmNodes".unitStatus.specialFunctions."Gauge R&R Type1" )
      I_Contact( #instTransferPnPLeftHomeJob1.jobStatus.active )
      I_Contact( #instTransferPnPLeftSideTapeLoadJob2.jobStatus.active )
      I_Contact( #instTransferPnPLeftHotPressLeftUnloadJob3.jobStatus.active )
      I_Contact( #instTransferPnPLeftHotPressLeftLoadJob4.jobStatus.active )
      I_Contact( #instTransferPnPLeftSideTapeLoadJob5.jobStatus.active )
      I_Contact( #instTransferPnPLeftHotPressRightUnloadJob6.jobStatus.active )
      I_Contact( #instTransferPnPLeftHotPressRightLoadJob7.jobStatus.active )
      I_Contact( #instTransferPnPLeftHipotThicknessUnloadJob9.jobStatus.active )
      I_Contact( #instTransferPnPRightHomeJob1.jobStatus.active )
      I_Contact( #instTransferPnPRightHipotThicknessLoadJob2.jobStatus.active )
      I_Contact( #instTransferPnPRightVisionUnloadJob3.jobStatus.active )
      I_Contact( #instTransferPnPRightVisionLoadJob4.jobStatus.active )
      I_Contact( #instTransferPnPRightLaserMarkUnloadJob5.jobStatus.active )
      I_Contact( #instTransferPnPRightLaserMarkLoadJob6.jobStatus.active )
      I_Contact( #instTransferPnPRightWeightCheckUnloadJob9.jobStatus.active )
   END_RUNG wire#w5
   RUNG wire#w4
      Contact( "Unit1.EmNodes".unitStatus.specialFunctions."Gauge R&R Type1" )
      I_Contact( #instGRnR_SideTapeLoadJob2_Left.jobStatus.active )
      I_Contact( #instGRnR_HipotThicknessUnloadJob3_Left.jobStatus.active )
      I_Contact( #instGRnR_HipotThicknessLoadJob4_Left.jobStatus.active )
      I_Contact( #instGRnR_HipotThicknessLoadJob5_Right.jobStatus.active )
      I_Contact( #instGRnR_VisionUnloadJob6_Right.jobStatus.active )
      I_Contact( #instGRnR_VisionLoadJob7_Right.jobStatus.active )
      I_Contact( #instGRnR_WeightCheckUnloadJob8_Right.jobStatus.active )
   END_RUNG wire#w5
   RUNG wire#powerrail
      Contact( #statUnitStatus.state.aborting )
      Contact( #TRUE )
   END_RUNG wire#w6
   RUNG wire#powerrail
      Contact( #statUnitStatus.state.clearing )
      Contact( #TRUE )
   END_RUNG wire#w7
   RUNG wire#powerrail
      Contact( #statUnitStatus.state.holding )
      Contact( #TRUE )
   END_RUNG wire#w8
   RUNG wire#powerrail
      Contact( #statUnitStatus.state.unholding )
      Contact( #TRUE )
   END_RUNG wire#w9
   RUNG wire#powerrail
      Contact( #statUnitStatus.state.suspending )
      Contact( #TRUE )
   END_RUNG wire#w10
   RUNG wire#powerrail
      Contact( #statUnitStatus.state.unsuspending )
      Contact( #TRUE )
   END_RUNG wire#w11
   RUNG wire#powerrail
      Contact( #statUnitStatus.state.completing )
      wire#w12
      I_Contact( "Unit1.EmNodes".unitStatus.specialFunctions."Gauge R&R Type1" )
      I_Contact( #instTransferPnPLeftHomeJob1.jobStatus.active )
      I_Contact( #instTransferPnPLeftSideTapeLoadJob2.jobStatus.active )
      I_Contact( #instTransferPnPLeftHotPressLeftUnloadJob3.jobStatus.active )
      I_Contact( #instTransferPnPLeftHotPressLeftLoadJob4.jobStatus.active )
      I_Contact( #instTransferPnPLeftSideTapeLoadJob5.jobStatus.active )
      I_Contact( #instTransferPnPLeftHotPressRightUnloadJob6.jobStatus.active )
      I_Contact( #instTransferPnPLeftHotPressRightLoadJob7.jobStatus.active )
      I_Contact( #instTransferPnPLeftHipotThicknessUnloadJob9.jobStatus.active )
      I_Contact( #instTransferPnPRightHomeJob1.jobStatus.active )
      I_Contact( #instTransferPnPRightHipotThicknessLoadJob2.jobStatus.active )
      I_Contact( #instTransferPnPRightVisionUnloadJob3.jobStatus.active )
      I_Contact( #instTransferPnPRightVisionLoadJob4.jobStatus.active )
      I_Contact( #instTransferPnPRightLaserMarkUnloadJob5.jobStatus.active )
      I_Contact( #instTransferPnPRightLaserMarkLoadJob6.jobStatus.active )
      I_Contact( #instTransferPnPRightWeightCheckUnloadJob9.jobStatus.active )
   END_RUNG wire#w13
   RUNG wire#w12
      Contact( "Unit1.EmNodes".unitStatus.specialFunctions."Gauge R&R Type1" )
      I_Contact( #instGRnR_SideTapeLoadJob2_Left.jobStatus.active )
      I_Contact( #instGRnR_HipotThicknessUnloadJob3_Left.jobStatus.active )
      I_Contact( #instGRnR_HipotThicknessLoadJob4_Left.jobStatus.active )
      I_Contact( #instGRnR_HipotThicknessLoadJob5_Right.jobStatus.active )
      I_Contact( #instGRnR_VisionUnloadJob6_Right.jobStatus.active )
      I_Contact( #instGRnR_VisionLoadJob7_Right.jobStatus.active )
      I_Contact( #instGRnR_WeightCheckUnloadJob8_Right.jobStatus.active )
   END_RUNG wire#w13
   // the same network as SCL:
   "LAF_DetermineStateComplete"(active := #statUnitStatus.mode.production,
                           resettingSC := #statUnitStatus.state.resetting AND NOT "Unit1.Em5.Alarms".emAlarms.error,
                           startingSC := #statUnitStatus.state.starting AND "Unit1.Em5.ControlNodes".em.status.initialized AND "Unit1.Em5.ControlNodes".em.status.homed AND "Unit1.EmNodes".stateCommandsExecute,
                           stoppingSC := #statUnitStatus.state.stopping AND ((NOT "Unit1.EmNodes".unitStatus.specialFunctions."Gauge R&R Type1" AND NOT #instTransferPnPLeftHomeJob1.jobStatus.active AND NOT #instTransferPnPLeftSideTapeLoadJob2.jobStatus.active AND NOT #instTransferPnPLeftHotPressLeftUnloadJob3.jobStatus.active AND NOT #instTransferPnPLeftHotPressLeftLoadJob4.jobStatus.active AND NOT #instTransferPnPLeftSideTapeLoadJob5.jobStatus.active AND NOT #instTransferPnPLeftHotPressRightUnloadJob6.jobStatus.active AND NOT #instTransferPnPLeftHotPressRightLoadJob7.jobStatus.active AND NOT #instTransferPnPLeftHipotThicknessUnloadJob9.jobStatus.active AND NOT #instTransferPnPRightHomeJob1.jobStatus.active AND NOT #instTransferPnPRightHipotThicknessLoadJob2.jobStatus.active AND NOT #instTransferPnPRightVisionUnloadJob3.jobStatus.active AND NOT #instTransferPnPRightVisionLoadJob4.jobStatus.active AND NOT #instTransferPnPRightLaserMarkUnloadJob5.jobStatus.active AND NOT #instTransferPnPRightLaserMarkLoadJob6.jobStatus.active AND NOT #instTransferPnPRightWeightCheckUnloadJob9.jobStatus.active) OR ("Unit1.EmNodes".unitStatus.specialFunctions."Gauge R&R Type1" AND NOT #instGRnR_SideTapeLoadJob2_Left.jobStatus.active AND NOT #instGRnR_HipotThicknessUnloadJob3_Left.jobStatus.active AND NOT #instGRnR_HipotThicknessLoadJob4_Left.jobStatus.active AND NOT #instGRnR_HipotThicknessLoadJob5_Right.jobStatus.active AND NOT #instGRnR_VisionUnloadJob6_Right.jobStatus.active AND NOT #instGRnR_VisionLoadJob7_Right.jobStatus.active AND NOT #instGRnR_WeightCheckUnloadJob8_Right.jobStatus.active)),
                           abortingSC := #statUnitStatus.state.aborting AND #TRUE,
                           clearingSC := #statUnitStatus.state.clearing AND #TRUE,
                           holdingSC := #statUnitStatus.state.holding AND #TRUE,
                           unholdingSC := #statUnitStatus.state.unholding AND #TRUE,
                           suspendingSC := #statUnitStatus.state.suspending AND #TRUE,
                           unsuspendingSC := #statUnitStatus.state.unsuspending AND #TRUE,
                           completingSC := #statUnitStatus.state.completing AND ((NOT "Unit1.EmNodes".unitStatus.specialFunctions."Gauge R&R Type1" AND NOT #instTransferPnPLeftHomeJob1.jobStatus.active AND NOT #instTransferPnPLeftSideTapeLoadJob2.jobStatus.active AND NOT #instTransferPnPLeftHotPressLeftUnloadJob3.jobStatus.active AND NOT #instTransferPnPLeftHotPressLeftLoadJob4.jobStatus.active AND NOT #instTransferPnPLeftSideTapeLoadJob5.jobStatus.active AND NOT #instTransferPnPLeftHotPressRightUnloadJob6.jobStatus.active AND NOT #instTransferPnPLeftHotPressRightLoadJob7.jobStatus.active AND NOT #instTransferPnPLeftHipotThicknessUnloadJob9.jobStatus.active AND NOT #instTransferPnPRightHomeJob1.jobStatus.active AND NOT #instTransferPnPRightHipotThicknessLoadJob2.jobStatus.active AND NOT #instTransferPnPRightVisionUnloadJob3.jobStatus.active AND NOT #instTransferPnPRightVisionLoadJob4.jobStatus.active AND NOT #instTransferPnPRightLaserMarkUnloadJob5.jobStatus.active AND NOT #instTransferPnPRightLaserMarkLoadJob6.jobStatus.active AND NOT #instTransferPnPRightWeightCheckUnloadJob9.jobStatus.active) OR ("Unit1.EmNodes".unitStatus.specialFunctions."Gauge R&R Type1" AND NOT #instGRnR_SideTapeLoadJob2_Left.jobStatus.active AND NOT #instGRnR_HipotThicknessUnloadJob3_Left.jobStatus.active AND NOT #instGRnR_HipotThicknessLoadJob4_Left.jobStatus.active AND NOT #instGRnR_HipotThicknessLoadJob5_Right.jobStatus.active AND NOT #instGRnR_VisionUnloadJob6_Right.jobStatus.active AND NOT #instGRnR_VisionLoadJob7_Right.jobStatus.active AND NOT #instGRnR_WeightCheckUnloadJob8_Right.jobStatus.active)),
                           stateComplete => #tempScInProduction);
END_REGION

REGION Network 220: Determine StateComplete (SC) in Mode Maintenance/Manual
   // Conditions for the Equipment Modules "stateComplete" feedback to the unit. This feedback is given when the task in for the respective state is complete.
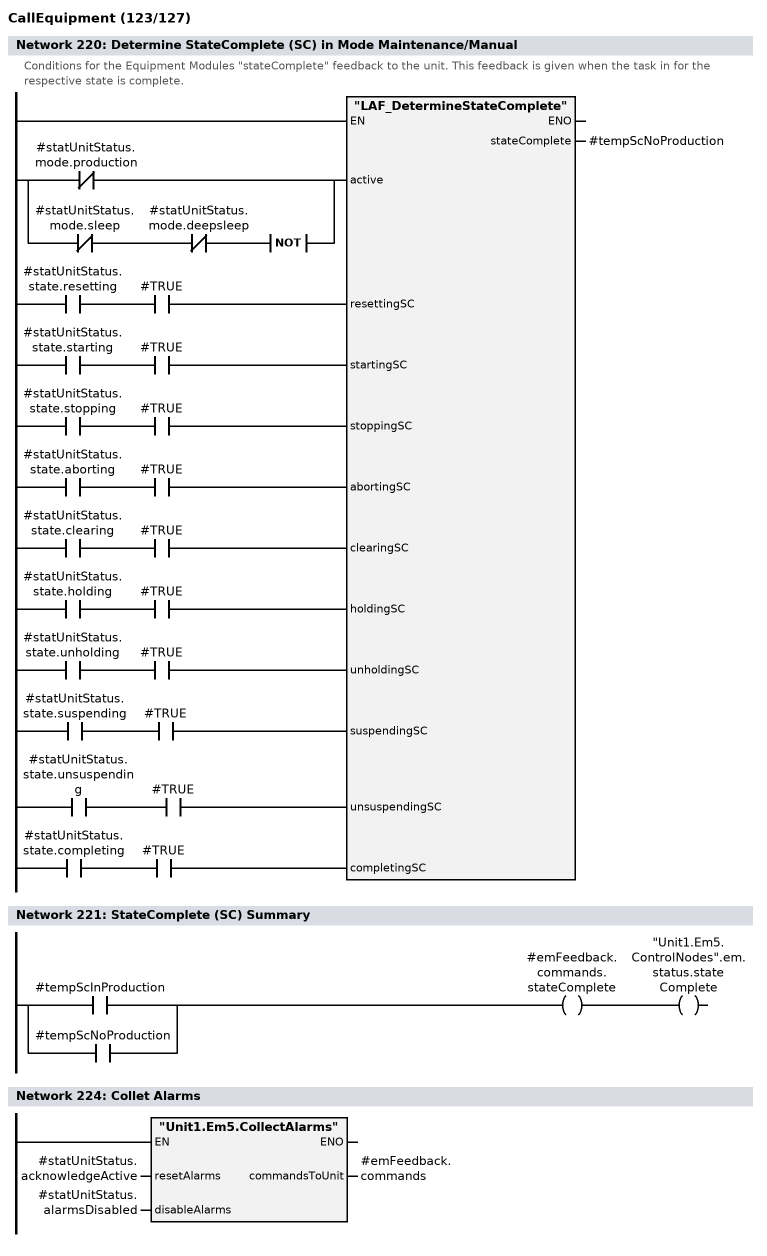
   RUNG wire#powerrail
      "LAF_DetermineStateComplete"(active := wire#w1, resettingSC := wire#w2, startingSC := wire#w3, stoppingSC := wire#w4, abortingSC := wire#w5, clearingSC := wire#w6, holdingSC := wire#w7, unholdingSC := wire#w8, suspendingSC := wire#w9, unsuspendingSC := wire#w10, completingSC := wire#w11, stateComplete => #tempScNoProduction)
   END_RUNG
   RUNG wire#powerrail
      I_Contact( #statUnitStatus.mode.production )
   END_RUNG wire#w1
   RUNG wire#powerrail
      I_Contact( #statUnitStatus.mode.sleep )
      I_Contact( #statUnitStatus.mode.deepsleep )
      Not()
   END_RUNG wire#w1
   RUNG wire#powerrail
      Contact( #statUnitStatus.state.resetting )
      Contact( #TRUE )
   END_RUNG wire#w2
   RUNG wire#powerrail
      Contact( #statUnitStatus.state.starting )
      Contact( #TRUE )
   END_RUNG wire#w3
   RUNG wire#powerrail
      Contact( #statUnitStatus.state.stopping )
      Contact( #TRUE )
   END_RUNG wire#w4
   RUNG wire#powerrail
      Contact( #statUnitStatus.state.aborting )
      Contact( #TRUE )
   END_RUNG wire#w5
   RUNG wire#powerrail
      Contact( #statUnitStatus.state.clearing )
      Contact( #TRUE )
   END_RUNG wire#w6
   RUNG wire#powerrail
      Contact( #statUnitStatus.state.holding )
      Contact( #TRUE )
   END_RUNG wire#w7
   RUNG wire#powerrail
      Contact( #statUnitStatus.state.unholding )
      Contact( #TRUE )
   END_RUNG wire#w8
   RUNG wire#powerrail
      Contact( #statUnitStatus.state.suspending )
      Contact( #TRUE )
   END_RUNG wire#w9
   RUNG wire#powerrail
      Contact( #statUnitStatus.state.unsuspending )
      Contact( #TRUE )
   END_RUNG wire#w10
   RUNG wire#powerrail
      Contact( #statUnitStatus.state.completing )
      Contact( #TRUE )
   END_RUNG wire#w11
   // the same network as SCL:
   "LAF_DetermineStateComplete"(active := NOT #statUnitStatus.mode.production OR NOT (NOT #statUnitStatus.mode.sleep AND NOT #statUnitStatus.mode.deepsleep),
                           resettingSC := #statUnitStatus.state.resetting AND #TRUE,
                           startingSC := #statUnitStatus.state.starting AND #TRUE,
                           stoppingSC := #statUnitStatus.state.stopping AND #TRUE,
                           abortingSC := #statUnitStatus.state.aborting AND #TRUE,
                           clearingSC := #statUnitStatus.state.clearing AND #TRUE,
                           holdingSC := #statUnitStatus.state.holding AND #TRUE,
                           unholdingSC := #statUnitStatus.state.unholding AND #TRUE,
                           suspendingSC := #statUnitStatus.state.suspending AND #TRUE,
                           unsuspendingSC := #statUnitStatus.state.unsuspending AND #TRUE,
                           completingSC := #statUnitStatus.state.completing AND #TRUE,
                           stateComplete => #tempScNoProduction);
END_REGION

REGION Network 221: StateComplete (SC) Summary
   RUNG wire#powerrail
      Contact( #tempScInProduction )
      wire#w1
      Coil( #emFeedback.commands.stateComplete )
      Coil( "Unit1.Em5.ControlNodes".em.status.stateComplete )
   END_RUNG
   RUNG wire#powerrail
      Contact( #tempScNoProduction )
   END_RUNG wire#w1
   // the same network as SCL:
   #emFeedback.commands.stateComplete := #tempScInProduction OR #tempScNoProduction;
   "Unit1.Em5.ControlNodes".em.status.stateComplete := #emFeedback.commands.stateComplete;
END_REGION

REGION Network 223: ******************** Alarms ********************
END_REGION

REGION Network 224: Collet Alarms
   RUNG wire#powerrail
      "Unit1.Em5.CollectAlarms"(resetAlarms := #statUnitStatus.acknowledgeActive, disableAlarms := #statUnitStatus.alarmsDisabled, commandsToUnit => #emFeedback.commands)
   END_RUNG
   // the same network as SCL:
   "Unit1.Em5.CollectAlarms"(resetAlarms := #statUnitStatus.acknowledgeActive,
                           disableAlarms := #statUnitStatus.alarmsDisabled,
                           commandsToUnit => #emFeedback.commands);
END_REGION

REGION Network 225: Manage Alarms
   // Derive commands from the ProDiag supervision. The ProDiag supervisions contain categories which define the reaction of these supervisions (e.g. abort, stop, hold). These are handed over as commands to the unit level.
   // Alternatively, if no ProDiag should be used, you can use the LAF_ManageBitAlarms to realize bit alarm handling. This block can be found in LAF in folder 70_AlarmHandling.
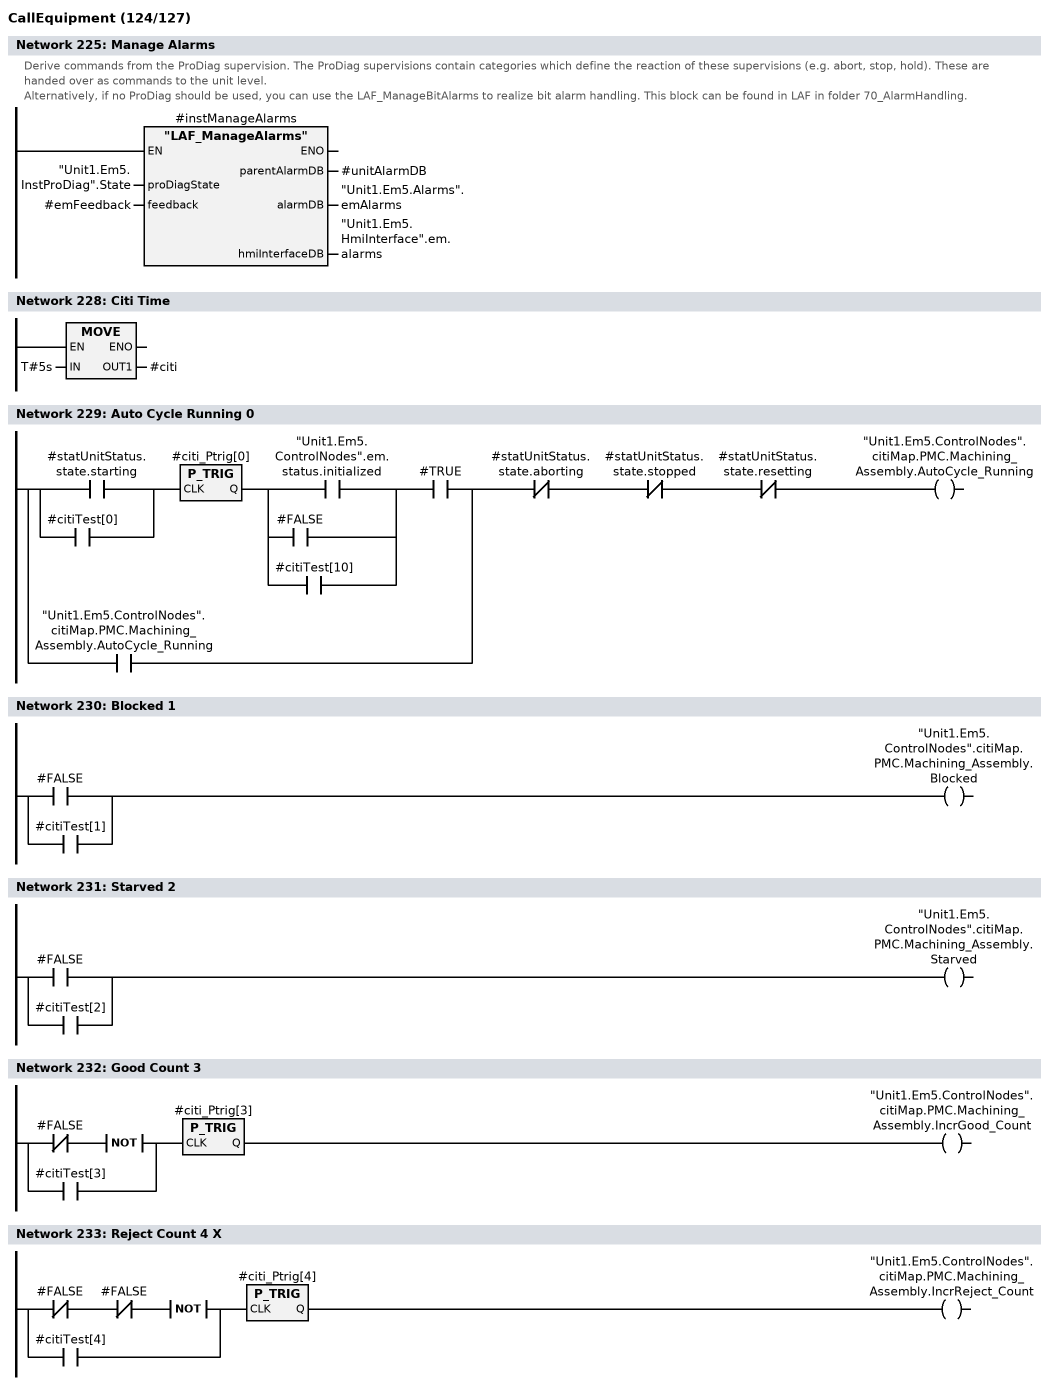
   RUNG wire#powerrail
      #instManageAlarms(proDiagState := "Unit1.Em5.InstProDiag".State, feedback := #emFeedback, parentAlarmDB => #unitAlarmDB, alarmDB => "Unit1.Em5.Alarms".emAlarms, hmiInterfaceDB => "Unit1.Em5.HmiInterface".em.alarms)
   END_RUNG
   // the same network as SCL:
   #instManageAlarms(proDiagState := "Unit1.Em5.InstProDiag".State,   // "LAF_ManageAlarms"
                     feedback := #emFeedback,
                     parentAlarmDB => #unitAlarmDB,
                     alarmDB => "Unit1.Em5.Alarms".emAlarms,
                     hmiInterfaceDB => "Unit1.Em5.HmiInterface".em.alarms);
END_REGION

REGION Network 227: ******************** CITI ********************
END_REGION

REGION Network 228: Citi Time
   RUNG wire#powerrail
      Move(in := T#5s, out1 => #citi)
   END_RUNG
   // the same network as SCL:
   #citi := T#5s;
END_REGION

REGION Network 229: Auto Cycle Running 0
   RUNG wire#powerrail
      Contact( #statUnitStatus.state.starting )
      wire#w1
      P_Trig( #citi_Ptrig[0] )
      wire#w2
      Contact( "Unit1.Em5.ControlNodes".em.status.initialized )
      wire#w3
      Contact( #TRUE )
      wire#w4
      I_Contact( #statUnitStatus.state.aborting )
      I_Contact( #statUnitStatus.state.stopped )
      I_Contact( #statUnitStatus.state.resetting )
      Coil( "Unit1.Em5.ControlNodes".citiMap.PMC.Machining_Assembly.AutoCycle_Running )
   END_RUNG
   RUNG wire#powerrail
      Contact( #citiTest[0] )
   END_RUNG wire#w1
   RUNG wire#w2
      Contact( #FALSE )
   END_RUNG wire#w3
   RUNG wire#w2
      Contact( #citiTest[10] )
   END_RUNG wire#w3
   RUNG wire#powerrail
      Contact( "Unit1.Em5.ControlNodes".citiMap.PMC.Machining_Assembly.AutoCycle_Running )
   END_RUNG wire#w4
   // the same network as SCL:
   #_w1 := #statUnitStatus.state.starting OR #citiTest[0];
   #_w2 := #_w1 AND NOT #citi_Ptrig[0];   // rising edge
   #citi_Ptrig[0] := #_w1;
   "Unit1.Em5.ControlNodes".citiMap.PMC.Machining_Assembly.AutoCycle_Running := ((#_w2 AND ("Unit1.Em5.ControlNodes".em.status.initialized OR #FALSE OR #citiTest[10]) AND #TRUE) OR "Unit1.Em5.ControlNodes".citiMap.PMC.Machining_Assembly.AutoCycle_Running) AND NOT #statUnitStatus.state.aborting AND NOT #statUnitStatus.state.stopped AND NOT #statUnitStatus.state.resetting;
END_REGION

REGION Network 230: Blocked 1
   RUNG wire#powerrail
      Contact( #FALSE )
      wire#w1
      Coil( "Unit1.Em5.ControlNodes".citiMap.PMC.Machining_Assembly.Blocked )
   END_RUNG
   RUNG wire#powerrail
      Contact( #citiTest[1] )
   END_RUNG wire#w1
   // the same network as SCL:
   "Unit1.Em5.ControlNodes".citiMap.PMC.Machining_Assembly.Blocked := #FALSE OR #citiTest[1];
END_REGION

REGION Network 231: Starved 2
   RUNG wire#powerrail
      Contact( #FALSE )
      wire#w1
      Coil( "Unit1.Em5.ControlNodes".citiMap.PMC.Machining_Assembly.Starved )
   END_RUNG
   RUNG wire#powerrail
      Contact( #citiTest[2] )
   END_RUNG wire#w1
   // the same network as SCL:
   "Unit1.Em5.ControlNodes".citiMap.PMC.Machining_Assembly.Starved := #FALSE OR #citiTest[2];
END_REGION

REGION Network 232: Good Count 3
   RUNG wire#powerrail
      I_Contact( #FALSE )
      Not()
      wire#w1
      P_Trig( #citi_Ptrig[3] )
      Coil( "Unit1.Em5.ControlNodes".citiMap.PMC.Machining_Assembly.IncrGood_Count )
   END_RUNG
   RUNG wire#powerrail
      Contact( #citiTest[3] )
   END_RUNG wire#w1
   // the same network as SCL:
   #_w1 := NOT (NOT #FALSE) OR #citiTest[3];
   #_w2 := #_w1 AND NOT #citi_Ptrig[3];   // rising edge
   #citi_Ptrig[3] := #_w1;
   "Unit1.Em5.ControlNodes".citiMap.PMC.Machining_Assembly.IncrGood_Count := #_w2;
END_REGION

REGION Network 233: Reject Count 4 X
   RUNG wire#powerrail
      I_Contact( #FALSE )
      I_Contact( #FALSE )
      Not()
      wire#w1
      P_Trig( #citi_Ptrig[4] )
      Coil( "Unit1.Em5.ControlNodes".citiMap.PMC.Machining_Assembly.IncrReject_Count )
   END_RUNG
   RUNG wire#powerrail
      Contact( #citiTest[4] )
   END_RUNG wire#w1
   // the same network as SCL:
   #_w1 := NOT (NOT #FALSE AND NOT #FALSE) OR #citiTest[4];
   #_w2 := #_w1 AND NOT #citi_Ptrig[4];   // rising edge
   #citi_Ptrig[4] := #_w1;
   "Unit1.Em5.ControlNodes".citiMap.PMC.Machining_Assembly.IncrReject_Count := #_w2;
END_REGION

REGION Network 234: Cycle End Trigger 5
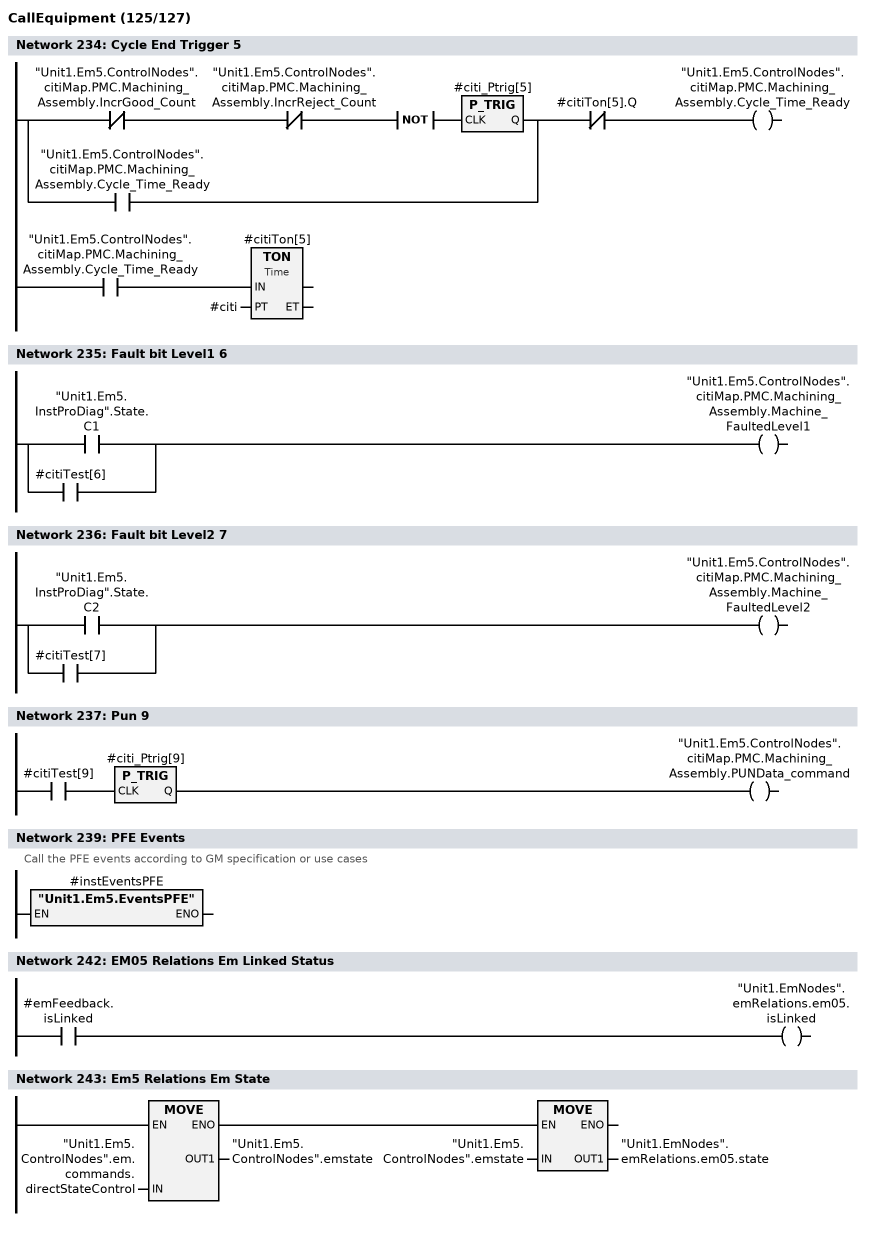
   RUNG wire#powerrail
      I_Contact( "Unit1.Em5.ControlNodes".citiMap.PMC.Machining_Assembly.IncrGood_Count )
      I_Contact( "Unit1.Em5.ControlNodes".citiMap.PMC.Machining_Assembly.IncrReject_Count )
      Not()
      P_Trig( #citi_Ptrig[5] )
      wire#w1
      I_Contact( #citiTon[5].Q )
      Coil( "Unit1.Em5.ControlNodes".citiMap.PMC.Machining_Assembly.Cycle_Time_Ready )
   END_RUNG
   RUNG wire#powerrail
      Contact( "Unit1.Em5.ControlNodes".citiMap.PMC.Machining_Assembly.Cycle_Time_Ready )
   END_RUNG wire#w1
   RUNG wire#powerrail
      Contact( "Unit1.Em5.ControlNodes".citiMap.PMC.Machining_Assembly.Cycle_Time_Ready )
      { S7_Templates := "time_type := Time" } #citiTon[5].TON(pt := #citi, et =>)
   END_RUNG
   // the same network as SCL:
   #_w1 := NOT (NOT "Unit1.Em5.ControlNodes".citiMap.PMC.Machining_Assembly.IncrGood_Count AND NOT "Unit1.Em5.ControlNodes".citiMap.PMC.Machining_Assembly.IncrReject_Count);
   #_w2 := #_w1 AND NOT #citi_Ptrig[5];   // rising edge
   #citi_Ptrig[5] := #_w1;
   "Unit1.Em5.ControlNodes".citiMap.PMC.Machining_Assembly.Cycle_Time_Ready := (#_w2 OR "Unit1.Em5.ControlNodes".citiMap.PMC.Machining_Assembly.Cycle_Time_Ready) AND NOT #citiTon[5].Q;
   #citiTon[5].TON(IN := "Unit1.Em5.ControlNodes".citiMap.PMC.Machining_Assembly.Cycle_Time_Ready, PT := #citi);
END_REGION

REGION Network 235: Fault bit Level1 6
   RUNG wire#powerrail
      Contact( "Unit1.Em5.InstProDiag".State.C1 )
      wire#w1
      Coil( "Unit1.Em5.ControlNodes".citiMap.PMC.Machining_Assembly.Machine_FaultedLevel1 )
   END_RUNG
   RUNG wire#powerrail
      Contact( #citiTest[6] )
   END_RUNG wire#w1
   // the same network as SCL:
   "Unit1.Em5.ControlNodes".citiMap.PMC.Machining_Assembly.Machine_FaultedLevel1 := "Unit1.Em5.InstProDiag".State.C1 OR #citiTest[6];
END_REGION

REGION Network 236: Fault bit Level2 7
   RUNG wire#powerrail
      Contact( "Unit1.Em5.InstProDiag".State.C2 )
      wire#w1
      Coil( "Unit1.Em5.ControlNodes".citiMap.PMC.Machining_Assembly.Machine_FaultedLevel2 )
   END_RUNG
   RUNG wire#powerrail
      Contact( #citiTest[7] )
   END_RUNG wire#w1
   // the same network as SCL:
   "Unit1.Em5.ControlNodes".citiMap.PMC.Machining_Assembly.Machine_FaultedLevel2 := "Unit1.Em5.InstProDiag".State.C2 OR #citiTest[7];
END_REGION

REGION Network 237: Pun 9
   RUNG wire#powerrail
      Contact( #citiTest[9] )
      P_Trig( #citi_Ptrig[9] )
      Coil( "Unit1.Em5.ControlNodes".citiMap.PMC.Machining_Assembly.PUNData_command )
   END_RUNG
   // the same network as SCL:
   #_w1 := #citiTest[9] AND NOT #citi_Ptrig[9];   // rising edge
   #citi_Ptrig[9] := #citiTest[9];
   "Unit1.Em5.ControlNodes".citiMap.PMC.Machining_Assembly.PUNData_command := #_w1;
END_REGION

REGION Network 238: ******************** PFE Events ********************
END_REGION

REGION Network 239: PFE Events
   // Call the PFE events according to GM specification or use cases
   RUNG wire#powerrail
      #instEventsPFE()
   END_RUNG
   // the same network as SCL:
   #instEventsPFE();   // "Unit1.Em5.EventsPFE"
END_REGION

REGION Network 241: ******************** Unit Output ********************
END_REGION

REGION Network 242: EM05 Relations Em Linked Status
   RUNG wire#powerrail
      Contact( #emFeedback.isLinked )
      Coil( "Unit1.EmNodes".emRelations.em05.isLinked )
   END_RUNG
   // the same network as SCL:
   "Unit1.EmNodes".emRelations.em05.isLinked := #emFeedback.isLinked;
END_REGION

REGION Network 243: Em5 Relations Em State
   RUNG wire#powerrail
      Move(in := "Unit1.Em5.ControlNodes".em.commands.directStateControl, out1 => "Unit1.Em5.ControlNodes".emstate)
      Move(in := "Unit1.Em5.ControlNodes".emstate, out1 => "Unit1.EmNodes".emRelations.em05.state)
   END_RUNG
   // the same network as SCL:
   "Unit1.Em5.ControlNodes".emstate := "Unit1.Em5.ControlNodes".em.commands.directStateControl;
   "Unit1.EmNodes".emRelations.em05.state := "Unit1.Em5.ControlNodes".emstate;
END_REGION

REGION Network 244: Em5 User define
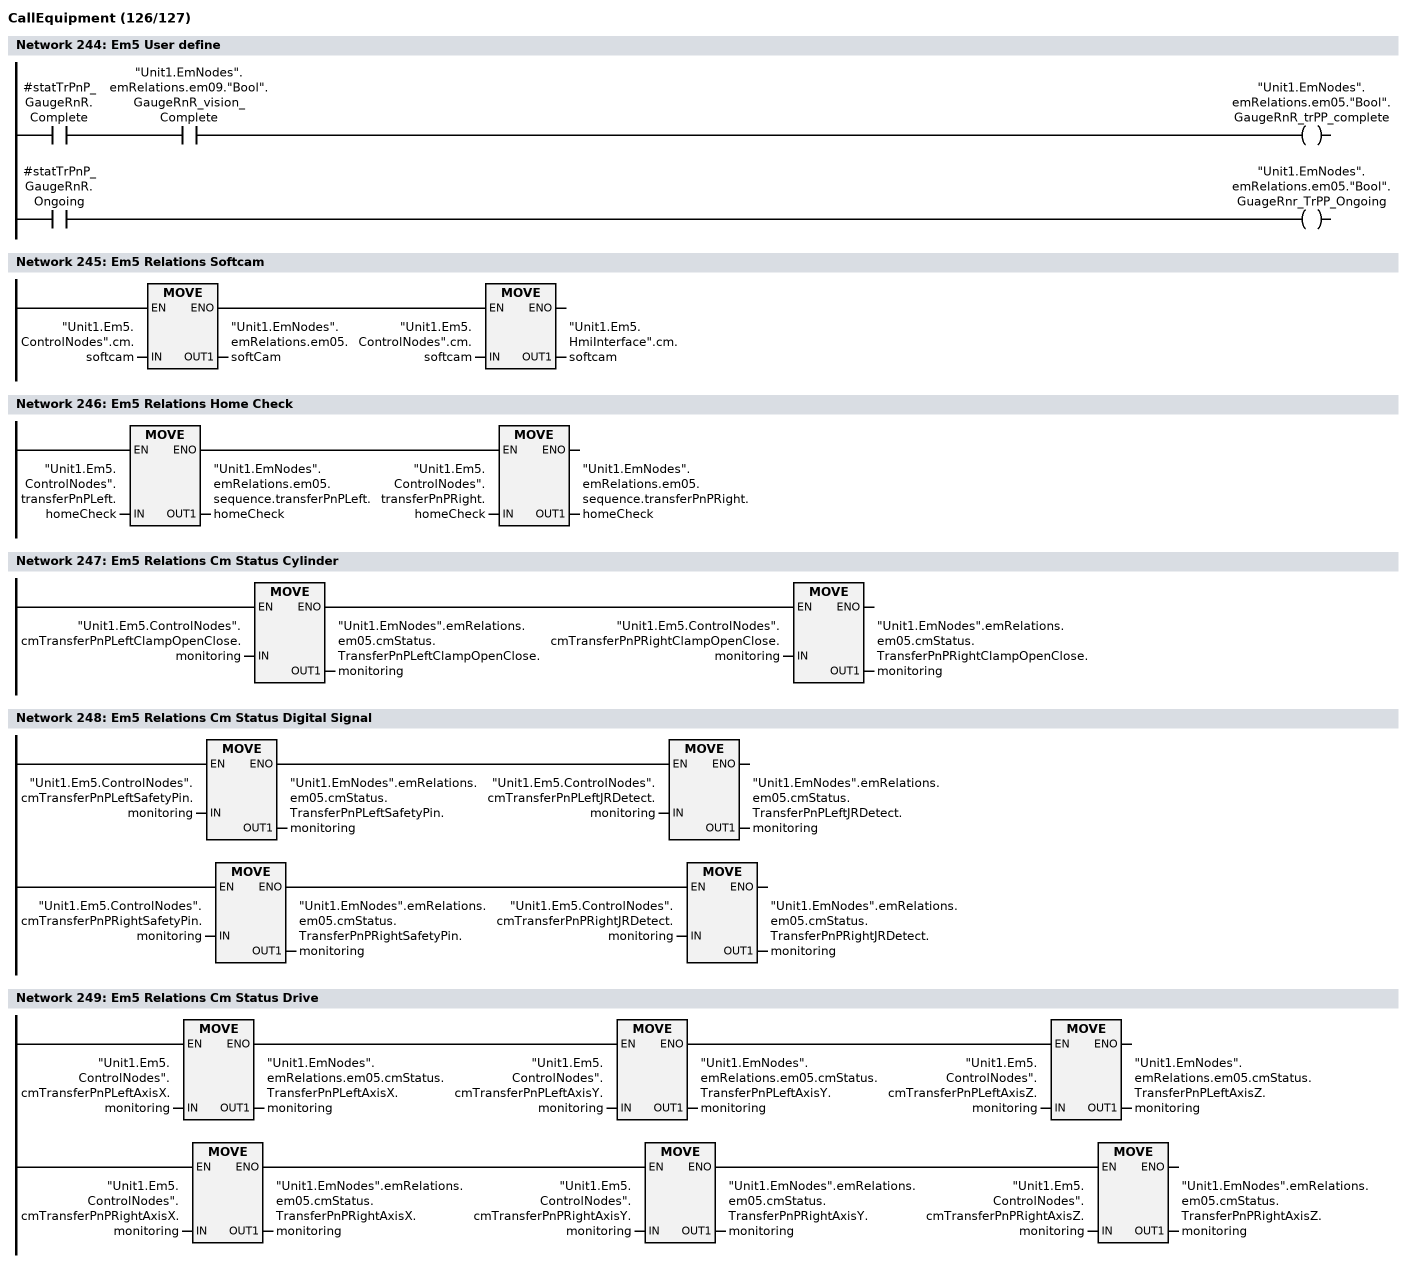
   RUNG wire#powerrail
      Contact( #statTrPnP_GaugeRnR.Complete )
      Contact( "Unit1.EmNodes".emRelations.em09."Bool".GaugeRnR_vision_Complete )
      Coil( "Unit1.EmNodes".emRelations.em05."Bool".GaugeRnR_trPP_complete )
   END_RUNG
   RUNG wire#powerrail
      Contact( #statTrPnP_GaugeRnR.Ongoing )
      Coil( "Unit1.EmNodes".emRelations.em05."Bool".GuageRnr_TrPP_Ongoing )
   END_RUNG
   // the same network as SCL:
   "Unit1.EmNodes".emRelations.em05."Bool".GaugeRnR_trPP_complete := #statTrPnP_GaugeRnR.Complete AND "Unit1.EmNodes".emRelations.em09."Bool".GaugeRnR_vision_Complete;
   "Unit1.EmNodes".emRelations.em05."Bool".GuageRnr_TrPP_Ongoing := #statTrPnP_GaugeRnR.Ongoing;
END_REGION

REGION Network 245: Em5 Relations Softcam
   RUNG wire#powerrail
      Move(in := "Unit1.Em5.ControlNodes".cm.softcam, out1 => "Unit1.EmNodes".emRelations.em05.softCam)
      Move(in := "Unit1.Em5.ControlNodes".cm.softcam, out1 => "Unit1.Em5.HmiInterface".cm.softcam)
   END_RUNG
   // the same network as SCL:
   "Unit1.EmNodes".emRelations.em05.softCam := "Unit1.Em5.ControlNodes".cm.softcam;
   "Unit1.Em5.HmiInterface".cm.softcam := "Unit1.Em5.ControlNodes".cm.softcam;
END_REGION

REGION Network 246: Em5 Relations Home Check
   RUNG wire#powerrail
      Move(in := "Unit1.Em5.ControlNodes".transferPnPLeft.homeCheck, out1 => "Unit1.EmNodes".emRelations.em05.sequence.transferPnPLeft.homeCheck)
      Move(in := "Unit1.Em5.ControlNodes".transferPnPRight.homeCheck, out1 => "Unit1.EmNodes".emRelations.em05.sequence.transferPnPRight.homeCheck)
   END_RUNG
   // the same network as SCL:
   "Unit1.EmNodes".emRelations.em05.sequence.transferPnPLeft.homeCheck := "Unit1.Em5.ControlNodes".transferPnPLeft.homeCheck;
   "Unit1.EmNodes".emRelations.em05.sequence.transferPnPRight.homeCheck := "Unit1.Em5.ControlNodes".transferPnPRight.homeCheck;
END_REGION

REGION Network 247: Em5 Relations Cm Status Cylinder
   RUNG wire#powerrail
      Move(in := "Unit1.Em5.ControlNodes".cmTransferPnPLeftClampOpenClose.monitoring, out1 => "Unit1.EmNodes".emRelations.em05.cmStatus.TransferPnPLeftClampOpenClose.monitoring)
      Move(in := "Unit1.Em5.ControlNodes".cmTransferPnPRightClampOpenClose.monitoring, out1 => "Unit1.EmNodes".emRelations.em05.cmStatus.TransferPnPRightClampOpenClose.monitoring)
   END_RUNG
   // the same network as SCL:
   "Unit1.EmNodes".emRelations.em05.cmStatus.TransferPnPLeftClampOpenClose.monitoring := "Unit1.Em5.ControlNodes".cmTransferPnPLeftClampOpenClose.monitoring;
   "Unit1.EmNodes".emRelations.em05.cmStatus.TransferPnPRightClampOpenClose.monitoring := "Unit1.Em5.ControlNodes".cmTransferPnPRightClampOpenClose.monitoring;
END_REGION

REGION Network 248: Em5 Relations Cm Status Digital Signal
   RUNG wire#powerrail
      Move(in := "Unit1.Em5.ControlNodes".cmTransferPnPLeftSafetyPin.monitoring, out1 => "Unit1.EmNodes".emRelations.em05.cmStatus.TransferPnPLeftSafetyPin.monitoring)
      Move(in := "Unit1.Em5.ControlNodes".cmTransferPnPLeftJRDetect.monitoring, out1 => "Unit1.EmNodes".emRelations.em05.cmStatus.TransferPnPLeftJRDetect.monitoring)
   END_RUNG
   RUNG wire#powerrail
      Move(in := "Unit1.Em5.ControlNodes".cmTransferPnPRightSafetyPin.monitoring, out1 => "Unit1.EmNodes".emRelations.em05.cmStatus.TransferPnPRightSafetyPin.monitoring)
      Move(in := "Unit1.Em5.ControlNodes".cmTransferPnPRightJRDetect.monitoring, out1 => "Unit1.EmNodes".emRelations.em05.cmStatus.TransferPnPRightJRDetect.monitoring)
   END_RUNG
   // the same network as SCL:
   "Unit1.EmNodes".emRelations.em05.cmStatus.TransferPnPLeftSafetyPin.monitoring := "Unit1.Em5.ControlNodes".cmTransferPnPLeftSafetyPin.monitoring;
   "Unit1.EmNodes".emRelations.em05.cmStatus.TransferPnPLeftJRDetect.monitoring := "Unit1.Em5.ControlNodes".cmTransferPnPLeftJRDetect.monitoring;
   "Unit1.EmNodes".emRelations.em05.cmStatus.TransferPnPRightSafetyPin.monitoring := "Unit1.Em5.ControlNodes".cmTransferPnPRightSafetyPin.monitoring;
   "Unit1.EmNodes".emRelations.em05.cmStatus.TransferPnPRightJRDetect.monitoring := "Unit1.Em5.ControlNodes".cmTransferPnPRightJRDetect.monitoring;
END_REGION

REGION Network 249: Em5 Relations Cm Status Drive
   RUNG wire#powerrail
      Move(in := "Unit1.Em5.ControlNodes".cmTransferPnPLeftAxisX.monitoring, out1 => "Unit1.EmNodes".emRelations.em05.cmStatus.TransferPnPLeftAxisX.monitoring)
      Move(in := "Unit1.Em5.ControlNodes".cmTransferPnPLeftAxisY.monitoring, out1 => "Unit1.EmNodes".emRelations.em05.cmStatus.TransferPnPLeftAxisY.monitoring)
      Move(in := "Unit1.Em5.ControlNodes".cmTransferPnPLeftAxisZ.monitoring, out1 => "Unit1.EmNodes".emRelations.em05.cmStatus.TransferPnPLeftAxisZ.monitoring)
   END_RUNG
   RUNG wire#powerrail
      Move(in := "Unit1.Em5.ControlNodes".cmTransferPnPRightAxisX.monitoring, out1 => "Unit1.EmNodes".emRelations.em05.cmStatus.TransferPnPRightAxisX.monitoring)
      Move(in := "Unit1.Em5.ControlNodes".cmTransferPnPRightAxisY.monitoring, out1 => "Unit1.EmNodes".emRelations.em05.cmStatus.TransferPnPRightAxisY.monitoring)
      Move(in := "Unit1.Em5.ControlNodes".cmTransferPnPRightAxisZ.monitoring, out1 => "Unit1.EmNodes".emRelations.em05.cmStatus.TransferPnPRightAxisZ.monitoring)
   END_RUNG
   // the same network as SCL:
   "Unit1.EmNodes".emRelations.em05.cmStatus.TransferPnPLeftAxisX.monitoring := "Unit1.Em5.ControlNodes".cmTransferPnPLeftAxisX.monitoring;
   "Unit1.EmNodes".emRelations.em05.cmStatus.TransferPnPLeftAxisY.monitoring := "Unit1.Em5.ControlNodes".cmTransferPnPLeftAxisY.monitoring;
   "Unit1.EmNodes".emRelations.em05.cmStatus.TransferPnPLeftAxisZ.monitoring := "Unit1.Em5.ControlNodes".cmTransferPnPLeftAxisZ.monitoring;
   "Unit1.EmNodes".emRelations.em05.cmStatus.TransferPnPRightAxisX.monitoring := "Unit1.Em5.ControlNodes".cmTransferPnPRightAxisX.monitoring;
   "Unit1.EmNodes".emRelations.em05.cmStatus.TransferPnPRightAxisY.monitoring := "Unit1.Em5.ControlNodes".cmTransferPnPRightAxisY.monitoring;
   "Unit1.EmNodes".emRelations.em05.cmStatus.TransferPnPRightAxisZ.monitoring := "Unit1.Em5.ControlNodes".cmTransferPnPRightAxisZ.monitoring;
END_REGION

REGION Network 250: Em5 Relations Sequence Interface
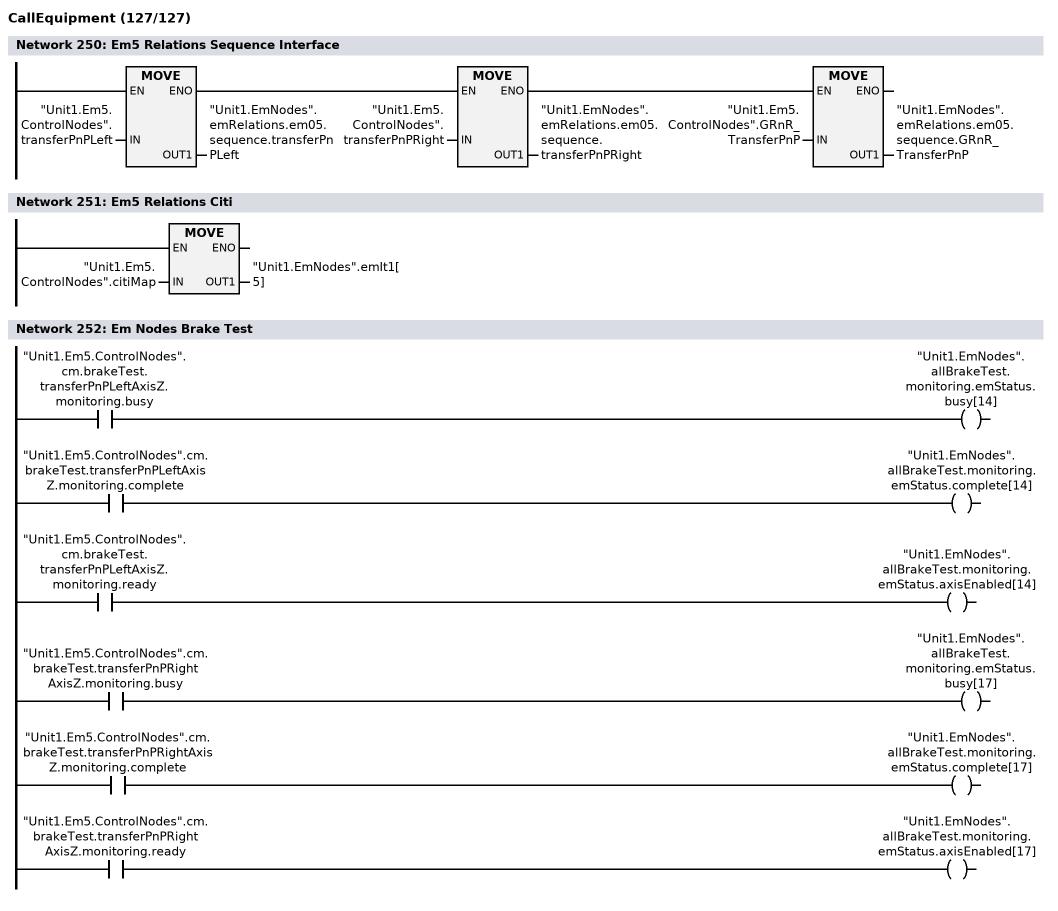
   RUNG wire#powerrail
      Move(in := "Unit1.Em5.ControlNodes".transferPnPLeft, out1 => "Unit1.EmNodes".emRelations.em05.sequence.transferPnPLeft)
      Move(in := "Unit1.Em5.ControlNodes".transferPnPRight, out1 => "Unit1.EmNodes".emRelations.em05.sequence.transferPnPRight)
      Move(in := "Unit1.Em5.ControlNodes".GRnR_TransferPnP, out1 => "Unit1.EmNodes".emRelations.em05.sequence.GRnR_TransferPnP)
   END_RUNG
   // the same network as SCL:
   "Unit1.EmNodes".emRelations.em05.sequence.transferPnPLeft := "Unit1.Em5.ControlNodes".transferPnPLeft;
   "Unit1.EmNodes".emRelations.em05.sequence.transferPnPRight := "Unit1.Em5.ControlNodes".transferPnPRight;
   "Unit1.EmNodes".emRelations.em05.sequence.GRnR_TransferPnP := "Unit1.Em5.ControlNodes".GRnR_TransferPnP;
END_REGION

REGION Network 251: Em5 Relations Citi
   RUNG wire#powerrail
      Move(in := "Unit1.Em5.ControlNodes".citiMap, out1 => "Unit1.EmNodes".emIt1[5])
   END_RUNG
   // the same network as SCL:
   "Unit1.EmNodes".emIt1[5] := "Unit1.Em5.ControlNodes".citiMap;
END_REGION

REGION Network 252: Em Nodes Brake Test
   RUNG wire#powerrail
      Contact( "Unit1.Em5.ControlNodes".cm.brakeTest.transferPnPLeftAxisZ.monitoring.busy )
      Coil( "Unit1.EmNodes".allBrakeTest.monitoring.emStatus.busy[14] )
   END_RUNG
   RUNG wire#powerrail
      Contact( "Unit1.Em5.ControlNodes".cm.brakeTest.transferPnPLeftAxisZ.monitoring.complete )
      Coil( "Unit1.EmNodes".allBrakeTest.monitoring.emStatus.complete[14] )
   END_RUNG
   RUNG wire#powerrail
      Contact( "Unit1.Em5.ControlNodes".cm.brakeTest.transferPnPLeftAxisZ.monitoring.ready )
      Coil( "Unit1.EmNodes".allBrakeTest.monitoring.emStatus.axisEnabled[14] )
   END_RUNG
   RUNG wire#powerrail
      Contact( "Unit1.Em5.ControlNodes".cm.brakeTest.transferPnPRightAxisZ.monitoring.busy )
      Coil( "Unit1.EmNodes".allBrakeTest.monitoring.emStatus.busy[17] )
   END_RUNG
   RUNG wire#powerrail
      Contact( "Unit1.Em5.ControlNodes".cm.brakeTest.transferPnPRightAxisZ.monitoring.complete )
      Coil( "Unit1.EmNodes".allBrakeTest.monitoring.emStatus.complete[17] )
   END_RUNG
   RUNG wire#powerrail
      Contact( "Unit1.Em5.ControlNodes".cm.brakeTest.transferPnPRightAxisZ.monitoring.ready )
      Coil( "Unit1.EmNodes".allBrakeTest.monitoring.emStatus.axisEnabled[17] )
   END_RUNG
   // the same network as SCL:
   "Unit1.EmNodes".allBrakeTest.monitoring.emStatus.busy[14] := "Unit1.Em5.ControlNodes".cm.brakeTest.transferPnPLeftAxisZ.monitoring.busy;
   "Unit1.EmNodes".allBrakeTest.monitoring.emStatus.complete[14] := "Unit1.Em5.ControlNodes".cm.brakeTest.transferPnPLeftAxisZ.monitoring.complete;
   "Unit1.EmNodes".allBrakeTest.monitoring.emStatus.axisEnabled[14] := "Unit1.Em5.ControlNodes".cm.brakeTest.transferPnPLeftAxisZ.monitoring.ready;
   "Unit1.EmNodes".allBrakeTest.monitoring.emStatus.busy[17] := "Unit1.Em5.ControlNodes".cm.brakeTest.transferPnPRightAxisZ.monitoring.busy;
   "Unit1.EmNodes".allBrakeTest.monitoring.emStatus.complete[17] := "Unit1.Em5.ControlNodes".cm.brakeTest.transferPnPRightAxisZ.monitoring.complete;
   "Unit1.EmNodes".allBrakeTest.monitoring.emStatus.axisEnabled[17] := "Unit1.Em5.ControlNodes".cm.brakeTest.transferPnPRightAxisZ.monitoring.ready;
END_REGION
END_FUNCTION_BLOCK
